C09139=1188.005,340.094,-74.713,-176.303,8.071,148.497
C09140=1188.000,340.372,-74.750,-176.301,8.074,148.497
C09141=1187.995,340.651,-74.787,-176.299,8.078,148.497
C09142=1187.991,340.929,-74.823,-176.296,8.081,148.498
C09143=1187.987,341.178,-74.856,-176.293,8.085,148.498
C09144=1187.982,341.425,-74.888,-176.291,8.088,148.498
C09145=1187.978,341.672,-74.921,-176.289,8.091,148.498
C09146=1187.974,341.921,-74.953,-176.287,8.094,148.498
C09147=1187.970,342.168,-74.987,-176.285,8.097,148.499
C09148=1187.966,342.416,-75.018,-176.283,8.101,148.499
C09149=1187.962,342.664,-75.052,-176.280,8.104,148.499
C09150=1187.958,342.912,-75.084,-176.278,8.107,148.499
C09151=1187.953,343.160,-75.117,-176.275,8.110,148.499
C09152=1187.950,343.408,-75.150,-176.273,8.114,148.499
C09153=1187.945,343.655,-75.182,-176.271,8.117,148.500
C09154=1187.941,343.903,-75.215,-176.269,8.120,148.500
C09155=1187.937,344.151,-75.248,-176.266,8.124,148.500
C09156=1187.932,344.399,-75.281,-176.264,8.127,148.500
C09157=1187.929,344.646,-75.313,-176.262,8.129,148.501
C09158=1187.925,344.894,-75.346,-176.260,8.133,148.501
C09159=1187.920,345.143,-75.379,-176.258,8.136,148.501
C09160=1187.916,345.390,-75.412,-176.256,8.139,148.501
C09161=1187.912,345.638,-75.445,-176.253,8.143,148.501
C09162=1187.909,345.885,-75.478,-176.251,8.146,148.502
C09163=1187.904,346.134,-75.510,-176.249,8.149,148.502
C09164=1187.900,346.382,-75.543,-176.247,8.153,148.502
C09165=1187.896,346.629,-75.576,-176.244,8.156,148.502
C09166=1187.892,346.877,-75.609,-176.242,8.159,148.502
C09167=1187.888,347.125,-75.643,-176.240,8.163,148.503
C09168=1187.883,347.373,-75.675,-176.238,8.165,148.503
C09169=1187.879,347.621,-75.708,-176.236,8.168,148.503
C09170=1187.876,347.868,-75.741,-176.234,8.172,148.503
C09171=1187.872,348.116,-75.774,-176.232,8.175,148.504
C09172=1187.867,348.364,-75.807,-176.229,8.178,148.504
C09173=1187.863,348.611,-75.840,-176.227,8.182,148.504
C09174=1187.859,348.859,-75.873,-176.225,8.185,148.504
C09175=1187.855,349.107,-75.907,-176.223,8.189,148.505
C09176=1187.851,349.355,-75.940,-176.221,8.192,148.505
C09177=1187.847,349.602,-75.973,-176.218,8.195,148.505
C09178=1187.842,349.851,-76.005,-176.216,8.199,148.505
C09179=1187.838,350.098,-76.038,-176.214,8.202,148.506
C09180=1187.834,350.346,-76.072,-176.212,8.205,148.506
C09181=1187.830,350.594,-76.105,-176.211,8.208,148.506
C09182=1187.826,350.842,-76.138,-176.208,8.211,148.506
C09183=1187.822,351.089,-76.171,-176.206,8.215,148.507
C09184=1187.818,351.336,-76.205,-176.204,8.218,148.507
C09185=1187.814,351.584,-76.238,-176.202,8.221,148.507
C09186=1187.809,351.832,-76.271,-176.200,8.225,148.507
C09187=1187.805,352.080,-76.304,-176.197,8.228,148.508
C09188=1187.801,352.327,-76.338,-176.195,8.232,148.508
C09189=1187.797,352.575,-76.371,-176.193,8.235,148.508
C09190=1187.793,352.824,-76.404,-176.191,8.238,148.508
C09191=1187.789,353.071,-76.437,-176.189,8.242,148.509
C09192=1187.785,353.319,-76.471,-176.187,8.245,148.509
C09193=1187.781,353.567,-76.504,-176.184,8.248,148.509
C09194=1187.777,353.814,-76.538,-176.183,8.251,148.510
C09195=1187.773,354.062,-76.571,-176.181,8.255,148.510
C09196=1187.768,354.310,-76.604,-176.179,8.258,148.510
C09197=1187.764,354.557,-76.638,-176.176,8.261,148.510
C09198=1187.760,354.805,-76.671,-176.175,8.265,148.511
C09199=1187.757,355.053,-76.705,-176.172,8.268,148.511
C09200=1187.753,355.301,-76.738,-176.170,8.272,148.511
C09201=1187.748,355.548,-76.771,-176.168,8.275,148.512
C09202=1187.744,355.796,-76.805,-176.166,8.278,148.512
C09203=1187.740,356.043,-76.838,-176.164,8.282,148.512
C09204=1187.736,356.291,-76.872,-176.162,8.285,148.512
C09205=1187.732,356.540,-76.906,-176.160,8.289,148.513
C09206=1187.728,356.787,-76.939,-176.158,8.292,148.513
C09207=1187.724,357.034,-76.973,-176.156,8.295,148.513
C09208=1187.720,357.282,-77.006,-176.154,8.298,148.513
C09209=1187.715,357.530,-77.040,-176.152,8.302,148.514
C09210=1187.711,357.777,-77.073,-176.150,8.305,148.514
C09211=1187.708,358.026,-77.107,-176.148,8.309,148.515
C09212=1187.704,358.273,-77.141,-176.146,8.312,148.515
C09213=1187.700,358.521,-77.174,-176.144,8.316,148.515
C09214=1187.695,358.769,-77.208,-176.142,8.319,148.515
C09215=1187.691,359.016,-77.242,-176.140,8.323,148.516
C09216=1187.687,359.264,-77.275,-176.138,8.326,148.516
C09217=1187.684,359.511,-77.309,-176.136,8.330,148.517
C09218=1187.679,359.759,-77.343,-176.134,8.333,148.517
C09219=1187.675,360.006,-77.377,-176.133,8.336,148.517
C09220=1187.671,360.255,-77.410,-176.131,8.339,148.518
C09221=1187.668,360.502,-77.444,-176.128,8.343,148.518
C09222=1187.663,360.750,-77.478,-176.127,8.346,148.518
C09223=1187.659,360.997,-77.512,-176.124,8.350,148.518
C09224=1187.655,361.246,-77.545,-176.123,8.353,148.519
C09225=1187.651,361.493,-77.580,-176.121,8.357,148.519
C09226=1187.647,361.741,-77.613,-176.119,8.359,148.520
C09227=1187.643,361.988,-77.647,-176.117,8.363,148.520
C09228=1187.639,362.236,-77.682,-176.116,8.367,148.520
C09229=1187.635,362.484,-77.715,-176.113,8.370,148.521
C09230=1187.631,362.731,-77.749,-176.111,8.374,148.521
C09231=1187.626,362.979,-77.782,-176.110,8.377,148.521
C09232=1187.623,363.227,-77.817,-176.108,8.380,148.522
C09233=1187.619,363.474,-77.850,-176.106,8.383,148.522
C09234=1187.614,363.722,-77.884,-176.104,8.387,148.523
C09235=1187.611,363.970,-77.918,-176.103,8.391,148.523
C09236=1187.606,364.217,-77.953,-176.101,8.394,148.523
C09237=1187.602,364.465,-77.986,-176.100,8.397,148.524
C09238=1187.599,364.713,-78.020,-176.098,8.401,148.524
C09239=1187.594,364.960,-78.055,-176.095,8.404,148.524
C09240=1187.590,365.208,-78.088,-176.094,8.408,148.525
C09241=1187.586,365.456,-78.123,-176.092,8.410,148.525
C09242=1187.582,365.703,-78.157,-176.091,8.414,148.526
C09243=1187.578,365.984,-78.195,-176.089,8.418,148.526
C09244=1187.573,366.265,-78.235,-176.086,8.422,148.527
C09245=1187.568,366.547,-78.273,-176.085,8.426,148.527
C09246=1187.564,366.828,-78.312,-176.083,8.429,148.527
C09247=1187.560,367.076,-78.345,-176.081,8.433,148.528
C09248=1187.556,367.323,-78.380,-176.079,8.437,148.528
C09249=1187.553,367.571,-78.414,-176.078,8.439,148.529
C09250=1187.548,367.819,-78.448,-176.076,8.443,148.529
C09251=1187.543,368.066,-78.482,-176.075,8.447,148.530
C09252=1187.540,368.314,-78.517,-176.074,8.450,148.530
C09253=1187.535,368.561,-78.551,-176.072,8.453,148.531
C09254=1187.532,368.809,-78.585,-176.070,8.457,148.531
C09255=1187.527,369.057,-78.620,-176.069,8.460,148.531
C09256=1187.524,369.304,-78.654,-176.067,8.463,148.532
C09257=1187.520,369.552,-78.688,-176.065,8.467,148.532
C09258=1187.516,369.799,-78.722,-176.064,8.470,148.533
C09259=1187.511,370.046,-78.757,-176.062,8.474,148.533
C09260=1187.508,370.295,-78.790,-176.061,8.477,148.534
C09261=1187.503,370.542,-78.825,-176.059,8.480,148.534
C09262=1187.499,370.790,-78.860,-176.058,8.484,148.535
C09263=1187.495,371.038,-78.893,-176.056,8.487,148.535
C09264=1187.491,371.286,-78.928,-176.055,8.490,148.536
C09265=1187.488,371.533,-78.962,-176.054,8.493,148.536
C09266=1187.483,371.780,-78.997,-176.052,8.497,148.536
C09267=1187.479,372.028,-79.031,-176.050,8.501,148.537
C09268=1187.475,372.275,-79.065,-176.049,8.504,148.537
C09269=1187.471,372.524,-79.100,-176.048,8.507,148.538
C09270=1187.467,372.770,-79.135,-176.046,8.510,148.538
C09271=1187.464,373.018,-79.170,-176.045,8.514,148.539
C09272=1187.459,373.266,-79.204,-176.044,8.517,148.539
C09273=1187.456,373.513,-79.238,-176.042,8.521,148.540
C09274=1187.451,373.761,-79.273,-176.041,8.523,148.540
C09275=1187.447,374.008,-79.307,-176.039,8.527,148.541
C09276=1187.443,374.256,-79.342,-176.039,8.530,148.541
C09277=1187.439,374.503,-79.376,-176.037,8.534,148.542
C09278=1187.435,374.752,-79.411,-176.036,8.537,148.542
C09279=1187.431,374.998,-79.446,-176.035,8.540,148.543
C09280=1187.428,375.246,-79.480,-176.033,8.544,148.543
C09281=1187.423,375.494,-79.515,-176.032,8.546,148.544
C09282=1187.419,375.742,-79.549,-176.031,8.550,148.544
C09283=1187.415,375.989,-79.583,-176.029,8.553,148.545
C09284=1187.411,376.237,-79.618,-176.029,8.556,148.545
C09285=1187.407,376.484,-79.653,-176.027,8.560,148.546
C09286=1187.403,376.732,-79.688,-176.026,8.563,148.546
C09287=1187.399,376.979,-79.722,-176.025,8.567,148.547
C09288=1187.395,377.227,-79.757,-176.023,8.570,148.547
C09289=1187.391,377.474,-79.792,-176.023,8.573,148.548
C09290=1187.387,377.722,-79.827,-176.021,8.576,148.548
C09291=1187.383,377.969,-79.861,-176.020,8.580,148.549
C09292=1187.379,378.217,-79.896,-176.019,8.583,148.550
C09293=1187.375,378.464,-79.931,-176.018,8.585,148.550
C09294=1187.371,378.712,-79.966,-176.017,8.589,148.551
C09295=1187.366,378.960,-80.000,-176.016,8.592,148.551
C09296=1187.363,379.207,-80.035,-176.015,8.595,148.552
C09297=1187.359,379.455,-80.070,-176.014,8.598,148.552
C09298=1187.355,379.702,-80.104,-176.012,8.602,148.553
C09299=1187.351,379.950,-80.139,-176.012,8.605,148.553
C09300=1187.347,380.197,-80.174,-176.011,8.608,148.554
C09301=1187.343,380.445,-80.209,-176.009,8.611,148.554
C09302=1187.339,380.692,-80.244,-176.009,8.614,148.555
C09303=1187.335,380.940,-80.279,-176.008,8.617,148.556
C09304=1187.331,381.187,-80.313,-176.007,8.621,148.556
C09305=1187.327,381.435,-80.349,-176.006,8.624,148.557
C09306=1187.322,381.682,-80.383,-176.004,8.627,148.557
C09307=1187.319,381.930,-80.419,-176.004,8.630,148.558
C09308=1187.315,382.178,-80.453,-176.003,8.633,148.558
C09309=1187.311,382.425,-80.487,-176.002,8.637,148.559
C09310=1187.307,382.673,-80.523,-176.001,8.640,148.559
C09311=1187.303,382.920,-80.557,-176.000,8.643,148.560
C09312=1187.299,383.167,-80.593,-176.000,8.646,148.561
C09313=1187.295,383.416,-80.628,-175.999,8.649,148.561
C09314=1187.291,383.662,-80.663,-175.998,8.652,148.562
C09315=1187.287,383.910,-80.698,-175.997,8.655,148.562
C09316=1187.283,384.157,-80.733,-175.996,8.658,148.563
C09317=1187.279,384.405,-80.767,-175.996,8.661,148.564
C09318=1187.276,384.653,-80.803,-175.995,8.664,148.564
C09319=1187.271,384.900,-80.837,-175.994,8.668,148.565
C09320=1187.267,385.148,-80.873,-175.993,8.671,148.565
C09321=1187.263,385.395,-80.907,-175.992,8.674,148.566
C09322=1187.259,385.642,-80.943,-175.992,8.677,148.566
C09323=1187.255,385.891,-80.978,-175.991,8.679,148.567
C09324=1187.251,386.137,-81.013,-175.991,8.682,148.568
C09325=1187.247,386.385,-81.048,-175.990,8.685,148.568
C09326=1187.243,386.632,-81.083,-175.989,8.688,148.569
C09327=1187.239,386.880,-81.118,-175.988,8.691,148.569
C09328=1187.235,387.128,-81.153,-175.988,8.694,148.570
C09329=1187.231,387.375,-81.188,-175.987,8.697,148.571
C09330=1187.227,387.623,-81.223,-175.987,8.700,148.571
C09331=1187.223,387.870,-81.259,-175.986,8.703,148.572
C09332=1187.219,388.118,-81.293,-175.986,8.706,148.572
C09333=1187.215,388.365,-81.329,-175.985,8.709,148.573
C09334=1187.211,388.613,-81.364,-175.984,8.712,148.574
C09335=1187.207,388.860,-81.399,-175.984,8.714,148.574
C09336=1187.203,389.108,-81.434,-175.983,8.717,148.575
C09337=1187.199,389.356,-81.469,-175.983,8.721,148.575
C09338=1187.195,389.603,-81.504,-175.982,8.723,148.576
C09339=1187.191,389.850,-81.540,-175.982,8.726,148.577
C09340=1187.187,390.098,-81.575,-175.981,8.729,148.577
C09341=1187.183,390.345,-81.610,-175.981,8.732,148.578
C09342=1187.179,390.592,-81.645,-175.980,8.735,148.578
C09343=1187.175,390.841,-81.680,-175.980,8.737,148.579
C09344=1187.171,391.087,-81.715,-175.979,8.740,148.580
C09345=1187.167,391.335,-81.751,-175.979,8.743,148.580
C09346=1187.164,391.582,-81.787,-175.978,8.746,148.581
C09347=1187.159,391.866,-81.827,-175.978,8.749,148.582
C09348=1187.155,392.150,-81.867,-175.978,8.751,148.582
C09349=1187.150,392.434,-81.907,-175.977,8.755,148.583
C09350=1187.145,392.717,-81.948,-175.977,8.758,148.584
C09351=1187.141,392.965,-81.983,-175.976,8.761,148.584
C09352=1187.137,393.212,-82.018,-175.976,8.764,148.585
C09353=1187.134,393.460,-82.054,-175.976,8.766,148.585
C09354=1187.129,393.706,-82.089,-175.975,8.769,148.586
C09355=1187.125,393.955,-82.124,-175.975,8.771,148.587
C09356=1187.122,394.202,-82.159,-175.974,8.775,148.587
C09357=1187.118,394.450,-82.195,-175.974,8.777,148.588
C09358=1187.114,394.696,-82.230,-175.974,8.779,148.588
C09359=1187.110,394.944,-82.265,-175.973,8.782,148.589
C09360=1187.106,395.192,-82.300,-175.973,8.785,148.590
C09361=1187.101,395.439,-82.336,-175.973,8.787,148.590
C09362=1187.097,395.687,-82.372,-175.973,8.790,148.591
C09363=1187.094,395.934,-82.407,-175.972,8.793,148.591
C09364=1187.090,396.182,-82.442,-175.973,8.795,148.592
C09365=1187.086,396.429,-82.477,-175.972,8.798,148.593
C09366=1187.082,396.676,-82.513,-175.972,8.800,148.593
C09367=1187.078,396.924,-82.548,-175.972,8.803,148.594
C09368=1187.074,397.171,-82.584,-175.971,8.805,148.595
C09369=1187.070,397.418,-82.619,-175.971,8.808,148.595
C09370=1187.066,397.667,-82.655,-175.971,8.810,148.596
C09371=1187.062,397.914,-82.690,-175.970,8.813,148.596
C09372=1187.058,398.161,-82.725,-175.970,8.816,148.597
C09373=1187.054,398.408,-82.761,-175.970,8.818,148.598
C09374=1187.050,398.656,-82.796,-175.970,8.820,148.598
C09375=1187.047,398.903,-82.832,-175.970,8.823,148.599
C09376=1187.042,399.150,-82.867,-175.970,8.825,148.599
C09377=1187.038,399.399,-82.903,-175.970,8.828,148.600
C09378=1187.034,399.646,-82.938,-175.969,8.831,148.600
C09379=1187.030,399.893,-82.973,-175.969,8.833,148.601
C09380=1187.026,400.141,-83.009,-175.969,8.835,148.602
C09381=1187.022,400.388,-83.044,-175.969,8.838,148.602
C09382=1187.019,400.636,-83.080,-175.968,8.840,148.603
C09383=1187.014,400.883,-83.116,-175.969,8.843,148.603
C09384=1187.010,401.130,-83.151,-175.968,8.845,148.604
C09385=1187.006,401.378,-83.187,-175.968,8.847,148.605
C09386=1187.003,401.625,-83.222,-175.968,8.850,148.605
C09387=1186.999,401.873,-83.257,-175.968,8.852,148.606
C09388=1186.994,402.120,-83.293,-175.968,8.854,148.606
C09389=1186.990,402.368,-83.329,-175.968,8.857,148.607
C09390=1186.986,402.615,-83.364,-175.968,8.859,148.608
C09391=1186.983,402.863,-83.400,-175.968,8.861,148.608
C09392=1186.979,403.110,-83.435,-175.967,8.864,148.609
C09393=1186.975,403.357,-83.470,-175.967,8.866,148.609
C09394=1186.970,403.605,-83.506,-175.967,8.868,148.610
C09395=1186.967,403.852,-83.542,-175.967,8.871,148.610
C09396=1186.963,404.099,-83.577,-175.967,8.873,148.611
C09397=1186.959,404.347,-83.613,-175.967,8.876,148.612
C09398=1186.954,404.595,-83.649,-175.967,8.878,148.612
C09399=1186.951,404.842,-83.684,-175.966,8.880,148.613
C09400=1186.947,405.090,-83.720,-175.967,8.883,148.613
C09401=1186.943,405.336,-83.755,-175.967,8.884,148.614
C09402=1186.939,405.584,-83.791,-175.967,8.886,148.614
C09403=1186.935,405.832,-83.827,-175.966,8.889,148.615
C09404=1186.931,406.079,-83.862,-175.967,8.891,148.616
C09405=1186.927,406.326,-83.898,-175.966,8.893,148.616
C09406=1186.923,406.573,-83.933,-175.966,8.896,148.617
C09407=1186.919,406.821,-83.969,-175.966,8.898,148.617
C09408=1186.915,407.069,-84.005,-175.967,8.900,148.618
C09409=1186.912,407.316,-84.040,-175.966,8.902,148.618
C09410=1186.907,407.563,-84.076,-175.966,8.904,148.619
C09411=1186.903,407.811,-84.112,-175.966,8.906,148.619
C09412=1186.899,408.058,-84.147,-175.966,8.909,148.620
C09413=1186.896,408.306,-84.183,-175.966,8.911,148.621
C09414=1186.892,408.553,-84.218,-175.966,8.913,148.621
C09415=1186.887,408.801,-84.254,-175.966,8.915,148.622
C09416=1186.883,409.048,-84.290,-175.965,8.917,148.622
C09417=1186.880,409.296,-84.325,-175.966,8.920,148.623
C09418=1186.876,409.542,-84.361,-175.966,8.921,148.623
C09419=1186.872,409.790,-84.398,-175.966,8.924,148.624
C09420=1186.868,410.038,-84.433,-175.965,8.926,148.624
C09421=1186.864,410.285,-84.468,-175.965,8.928,148.625
C09422=1186.860,410.532,-84.504,-175.966,8.930,148.625
C09423=1186.856,410.780,-84.540,-175.966,8.932,148.626
C09424=1186.852,411.027,-84.576,-175.965,8.934,148.627
C09425=1186.848,411.275,-84.611,-175.965,8.937,148.627
C09426=1186.843,411.522,-84.647,-175.965,8.938,148.628
C09427=1186.840,411.769,-84.682,-175.965,8.940,148.628
C09428=1186.836,412.017,-84.718,-175.965,8.943,148.629
C09429=1186.832,412.264,-84.754,-175.966,8.944,148.629
C09430=1186.828,412.512,-84.790,-175.965,8.947,148.630
C09431=1186.825,412.759,-84.826,-175.965,8.949,148.630
C09432=1186.820,413.006,-84.861,-175.966,8.950,148.631
C09433=1186.816,413.254,-84.897,-175.965,8.953,148.631
C09434=1186.812,413.501,-84.933,-175.965,8.955,148.632
C09435=1186.809,413.749,-84.968,-175.965,8.957,148.632
C09436=1186.804,413.997,-85.005,-175.965,8.958,148.633
C09437=1186.801,414.244,-85.040,-175.965,8.961,148.633
C09438=1186.797,414.490,-85.076,-175.965,8.962,148.634
C09439=1186.793,414.738,-85.112,-175.965,8.964,148.634
C09440=1186.789,414.986,-85.148,-175.965,8.967,148.635
C09441=1186.785,415.233,-85.183,-175.965,8.968,148.636
C09442=1186.781,415.481,-85.219,-175.965,8.971,148.636
C09443=1186.774,415.892,-85.279,-175.965,8.974,148.637
C09444=1186.770,416.304,-85.338,-175.965,8.977,148.638
C09445=1186.770,416.715,-85.397,-175.964,8.980,148.638
C09446=1186.774,417.125,-85.456,-175.965,8.983,148.639
C09447=1186.353,417.127,-85.497,-175.968,8.994,148.643
C09448=1186.349,416.714,-85.438,-175.968,8.991,148.642
C09449=1186.349,416.299,-85.379,-175.968,8.988,148.641
C09450=1186.353,415.883,-85.319,-175.968,8.985,148.640
C09451=1186.360,415.469,-85.259,-175.968,8.981,148.640
C09452=1186.363,415.222,-85.223,-175.968,8.979,148.639
C09453=1186.368,414.974,-85.187,-175.968,8.978,148.639
C09454=1186.371,414.727,-85.151,-175.968,8.975,148.638
C09455=1186.375,414.480,-85.116,-175.968,8.974,148.638
C09456=1186.380,414.232,-85.080,-175.968,8.971,148.637
C09457=1186.383,413.985,-85.044,-175.968,8.969,148.636
C09458=1186.387,413.737,-85.008,-175.968,8.968,148.636
C09459=1186.391,413.490,-84.972,-175.968,8.965,148.636
C09460=1186.395,413.243,-84.936,-175.968,8.963,148.635
C09461=1186.399,412.996,-84.901,-175.968,8.962,148.635
C09462=1186.403,412.748,-84.865,-175.968,8.959,148.634
C09463=1186.407,412.501,-84.829,-175.968,8.957,148.633
C09464=1186.411,412.253,-84.794,-175.968,8.956,148.633
C09465=1186.414,412.006,-84.758,-175.968,8.953,148.632
C09466=1186.419,411.758,-84.722,-175.968,8.951,148.632
C09467=1186.423,411.511,-84.687,-175.969,8.949,148.631
C09468=1186.427,411.264,-84.651,-175.968,8.947,148.631
C09469=1186.431,411.016,-84.614,-175.968,8.945,148.630
C09470=1186.435,410.769,-84.579,-175.969,8.943,148.630
C09471=1186.438,410.521,-84.543,-175.968,8.941,148.629
C09472=1186.443,410.274,-84.507,-175.968,8.939,148.629
C09473=1186.447,410.027,-84.472,-175.969,8.936,148.628
C09474=1186.451,409.779,-84.436,-175.969,8.934,148.628
C09475=1186.454,409.532,-84.401,-175.968,8.933,148.627
C09476=1186.459,409.284,-84.365,-175.969,8.931,148.627
C09477=1186.462,409.036,-84.329,-175.969,8.928,148.626
C09478=1186.466,408.790,-84.294,-175.969,8.926,148.625
C09479=1186.470,408.542,-84.258,-175.968,8.924,148.625
C09480=1186.475,408.294,-84.222,-175.969,8.922,148.624
C09481=1186.478,408.047,-84.186,-175.969,8.920,148.624
C09482=1186.482,407.800,-84.150,-175.969,8.917,148.623
C09483=1186.486,407.553,-84.115,-175.969,8.915,148.623
C09484=1186.490,407.305,-84.079,-175.969,8.913,148.622
C09485=1186.494,407.058,-84.044,-175.969,8.911,148.622
C09486=1186.498,406.810,-84.008,-175.969,8.909,148.621
C09487=1186.501,406.563,-83.972,-175.969,8.906,148.620
C09488=1186.506,406.316,-83.937,-175.969,8.904,148.620
C09489=1186.510,406.068,-83.901,-175.970,8.902,148.619
C09490=1186.514,405.821,-83.866,-175.969,8.900,148.619
C09491=1186.517,405.573,-83.830,-175.969,8.898,148.618
C09492=1186.522,405.325,-83.794,-175.969,8.896,148.618
C09493=1186.526,405.079,-83.759,-175.970,8.893,148.617
C09494=1186.530,404.831,-83.723,-175.969,8.891,148.616
C09495=1186.533,404.584,-83.688,-175.970,8.888,148.616
C09496=1186.537,404.336,-83.652,-175.970,8.886,148.615
C09497=1186.541,404.088,-83.616,-175.970,8.884,148.615
C09498=1186.546,403.842,-83.581,-175.970,8.881,148.614
C09499=1186.549,403.594,-83.545,-175.970,8.879,148.614
C09500=1186.553,403.346,-83.510,-175.970,8.877,148.613
C09501=1186.557,403.099,-83.474,-175.970,8.874,148.612
C09502=1186.562,402.852,-83.438,-175.970,8.873,148.612
C09503=1186.565,402.604,-83.403,-175.970,8.871,148.611
C09504=1186.569,402.357,-83.367,-175.970,8.868,148.611
C09505=1186.573,402.109,-83.332,-175.970,8.866,148.610
C09506=1186.578,401.862,-83.296,-175.971,8.863,148.609
C09507=1186.581,401.614,-83.261,-175.970,8.861,148.609
C09508=1186.585,401.367,-83.226,-175.971,8.859,148.608
C09509=1186.589,401.119,-83.190,-175.972,8.856,148.608
C09510=1186.592,400.872,-83.154,-175.971,8.853,148.607
C09511=1186.597,400.625,-83.119,-175.972,8.851,148.606
C09512=1186.601,400.377,-83.083,-175.972,8.848,148.606
C09513=1186.605,400.130,-83.048,-175.972,8.846,148.605
C09514=1186.608,399.882,-83.012,-175.972,8.844,148.605
C09515=1186.613,399.635,-82.977,-175.972,8.841,148.604
C09516=1186.616,399.388,-82.941,-175.972,8.839,148.603
C09517=1186.620,399.140,-82.906,-175.972,8.837,148.603
C09518=1186.625,398.892,-82.870,-175.972,8.834,148.602
C09519=1186.629,398.645,-82.835,-175.972,8.832,148.602
C09520=1186.633,398.398,-82.800,-175.973,8.829,148.601
C09521=1186.636,398.150,-82.764,-175.973,8.826,148.601
C09522=1186.640,397.903,-82.729,-175.973,8.824,148.600
C09523=1186.644,397.656,-82.693,-175.973,8.821,148.599
C09524=1186.649,397.408,-82.657,-175.974,8.819,148.599
C09525=1186.652,397.160,-82.622,-175.973,8.817,148.598
C09526=1186.657,396.913,-82.587,-175.974,8.814,148.597
C09527=1186.661,396.665,-82.552,-175.975,8.811,148.597
C09528=1186.664,396.418,-82.516,-175.974,8.809,148.596
C09529=1186.668,396.170,-82.481,-175.975,8.806,148.596
C09530=1186.672,395.924,-82.445,-175.975,8.803,148.595
C09531=1186.676,395.676,-82.411,-175.975,8.801,148.594
C09532=1186.681,395.428,-82.374,-175.975,8.799,148.594
C09533=1186.685,395.181,-82.339,-175.976,8.795,148.593
C09534=1186.688,394.933,-82.304,-175.976,8.793,148.593
C09535=1186.692,394.686,-82.268,-175.976,8.791,148.592
C09536=1186.696,394.438,-82.233,-175.977,8.787,148.591
C09537=1186.700,394.191,-82.198,-175.977,8.785,148.591
C09538=1186.704,393.944,-82.163,-175.977,8.783,148.590
C09539=1186.708,393.696,-82.127,-175.978,8.780,148.590
C09540=1186.712,393.449,-82.092,-175.978,8.777,148.589
C09541=1186.716,393.201,-82.057,-175.978,8.775,148.588
C09542=1186.720,392.954,-82.021,-175.979,8.772,148.588
C09543=1186.723,392.706,-81.986,-175.979,8.769,148.587
C09544=1186.728,392.422,-81.946,-175.980,8.766,148.586
C09545=1186.732,392.139,-81.905,-175.980,8.763,148.586
C09546=1186.737,391.855,-81.865,-175.981,8.759,148.585
C09547=1186.742,391.571,-81.824,-175.981,8.756,148.584
C09548=1186.746,391.325,-81.789,-175.981,8.754,148.584
C09549=1186.750,391.076,-81.754,-175.982,8.751,148.583
C09550=1186.754,390.829,-81.718,-175.982,8.748,148.582
C09551=1186.758,390.582,-81.683,-175.983,8.745,148.582
C09552=1186.762,390.334,-81.648,-175.983,8.743,148.581
C09553=1186.766,390.086,-81.612,-175.984,8.740,148.581
C09554=1186.770,389.839,-81.577,-175.984,8.737,148.580
C09555=1186.774,389.591,-81.542,-175.984,8.734,148.579
C09556=1186.778,389.344,-81.507,-175.985,8.731,148.579
C09557=1186.782,389.097,-81.472,-175.985,8.729,148.578
C09558=1186.786,388.849,-81.437,-175.986,8.725,148.578
C09559=1186.790,388.601,-81.401,-175.987,8.722,148.577
C09560=1186.794,388.355,-81.366,-175.987,8.720,148.576
C09561=1186.798,388.106,-81.331,-175.988,8.717,148.576
C09562=1186.802,387.859,-81.296,-175.989,8.714,148.575
C09563=1186.806,387.612,-81.261,-175.988,8.711,148.575
C09564=1186.810,387.364,-81.226,-175.989,8.708,148.574
C09565=1186.814,387.117,-81.190,-175.990,8.705,148.573
C09566=1186.818,386.869,-81.156,-175.991,8.702,148.573
C09567=1186.821,386.622,-81.121,-175.991,8.700,148.572
C09568=1186.825,386.374,-81.086,-175.992,8.696,148.572
C09569=1186.829,386.127,-81.051,-175.993,8.693,148.571
C09570=1186.833,385.879,-81.015,-175.993,8.690,148.571
C09571=1186.838,385.632,-80.981,-175.994,8.687,148.570
C09572=1186.841,385.385,-80.945,-175.995,8.684,148.569
C09573=1186.845,385.136,-80.910,-175.995,8.681,148.569
C09574=1186.849,384.890,-80.875,-175.996,8.678,148.568
C09575=1186.853,384.642,-80.840,-175.996,8.675,148.567
C09576=1186.857,384.394,-80.805,-175.997,8.672,148.567
C09577=1186.862,384.147,-80.770,-175.998,8.669,148.566
C09578=1186.865,383.899,-80.735,-175.999,8.666,148.566
C09579=1186.870,383.652,-80.700,-176.000,8.663,148.565
C09580=1186.874,383.404,-80.665,-176.001,8.660,148.565
C09581=1186.878,383.156,-80.630,-176.001,8.657,148.564
C09582=1186.881,382.910,-80.595,-176.002,8.654,148.563
C09583=1186.885,382.661,-80.561,-176.003,8.651,148.563
C09584=1186.889,382.415,-80.525,-176.004,8.648,148.562
C09585=1186.893,382.167,-80.491,-176.005,8.645,148.562
C09586=1186.898,381.919,-80.456,-176.006,8.642,148.561
C09587=1186.902,381.672,-80.421,-176.007,8.638,148.561
C09588=1186.905,381.423,-80.386,-176.008,8.635,148.560
C09589=1186.910,381.177,-80.351,-176.009,8.631,148.559
C09590=1186.913,380.929,-80.316,-176.010,8.628,148.559
C09591=1186.918,380.681,-80.282,-176.011,8.626,148.558
C09592=1186.921,380.434,-80.246,-176.012,8.622,148.558
C09593=1186.926,380.187,-80.212,-176.012,8.619,148.557
C09594=1186.929,379.939,-80.176,-176.014,8.615,148.557
C09595=1186.933,379.691,-80.141,-176.015,8.612,148.556
C09596=1186.937,379.444,-80.108,-176.016,8.610,148.556
C09597=1186.941,379.196,-80.072,-176.017,8.606,148.555
C09598=1186.945,378.949,-80.038,-176.018,8.603,148.554
C09599=1186.949,378.701,-80.003,-176.019,8.599,148.554
C09600=1186.954,378.454,-79.968,-176.020,8.597,148.554
C09601=1186.957,378.206,-79.933,-176.021,8.594,148.553
C09602=1186.962,377.959,-79.899,-176.022,8.590,148.552
C09603=1186.965,377.711,-79.864,-176.024,8.587,148.552
C09604=1186.970,377.464,-79.829,-176.024,8.584,148.551
C09605=1186.974,377.216,-79.794,-176.026,8.580,148.551
C09606=1186.978,376.969,-79.760,-176.027,8.577,148.550
C09607=1186.982,376.720,-79.725,-176.028,8.574,148.550
C09608=1186.986,376.474,-79.690,-176.030,8.570,148.549
C09609=1186.990,376.226,-79.655,-176.030,8.567,148.549
C09610=1186.994,375.978,-79.621,-176.032,8.564,148.548
C09611=1186.998,375.730,-79.587,-176.033,8.560,148.548
C09612=1187.002,375.483,-79.552,-176.034,8.557,148.547
C09613=1187.005,375.236,-79.517,-176.036,8.554,148.547
C09614=1187.010,374.988,-79.483,-176.036,8.551,148.546
C09615=1187.014,374.740,-79.448,-176.038,8.547,148.546
C09616=1187.018,374.493,-79.413,-176.039,8.544,148.545
C09617=1187.021,374.245,-79.379,-176.040,8.541,148.545
C09618=1187.026,373.998,-79.345,-176.042,8.538,148.544
C09619=1187.030,373.750,-79.309,-176.043,8.534,148.544
C09620=1187.033,373.503,-79.275,-176.045,8.531,148.543
C09621=1187.037,373.255,-79.240,-176.045,8.528,148.543
C09622=1187.042,373.007,-79.206,-176.047,8.524,148.542
C09623=1187.045,372.760,-79.172,-176.049,8.521,148.542
C09624=1187.050,372.512,-79.137,-176.050,8.517,148.541
C09625=1187.054,372.265,-79.103,-176.052,8.514,148.541
C09626=1187.058,372.017,-79.069,-176.053,8.511,148.540
C09627=1187.062,371.770,-79.034,-176.054,8.507,148.540
C09628=1187.065,371.522,-79.000,-176.056,8.504,148.539
C09629=1187.070,371.274,-78.965,-176.057,8.501,148.539
C09630=1187.074,371.026,-78.931,-176.058,8.497,148.538
C09631=1187.078,370.779,-78.897,-176.060,8.494,148.538
C09632=1187.082,370.532,-78.862,-176.062,8.490,148.537
C09633=1187.086,370.284,-78.828,-176.063,8.487,148.537
C09634=1187.090,370.036,-78.793,-176.065,8.484,148.537
C09635=1187.094,369.788,-78.759,-176.066,8.481,148.536
C09636=1187.098,369.541,-78.725,-176.067,8.477,148.536
C09637=1187.102,369.294,-78.690,-176.069,8.473,148.535
C09638=1187.106,369.046,-78.656,-176.070,8.471,148.535
C09639=1187.110,368.799,-78.622,-176.072,8.467,148.534
C09640=1187.114,368.551,-78.587,-176.074,8.463,148.534
C09641=1187.118,368.303,-78.553,-176.075,8.461,148.534
C09642=1187.122,368.056,-78.520,-176.077,8.457,148.533
C09643=1187.126,367.807,-78.485,-176.079,8.453,148.533
C09644=1187.130,367.560,-78.451,-176.080,8.449,148.532
C09645=1187.135,367.313,-78.417,-176.082,8.447,148.532
C09646=1187.138,367.065,-78.382,-176.083,8.443,148.531
C09647=1187.142,366.818,-78.348,-176.085,8.439,148.531
C09648=1187.147,366.536,-78.310,-176.087,8.436,148.530
C09649=1187.151,366.254,-78.271,-176.089,8.432,148.530
C09650=1187.156,365.973,-78.232,-176.091,8.429,148.529
C09651=1187.161,365.692,-78.193,-176.093,8.424,148.529
C09652=1187.164,365.445,-78.159,-176.094,8.421,148.529
C09653=1187.169,365.196,-78.125,-176.096,8.418,148.528
C09654=1187.173,364.949,-78.091,-176.098,8.414,148.528
C09655=1187.177,364.702,-78.057,-176.100,8.411,148.528
C09656=1187.180,364.454,-78.022,-176.102,8.407,148.527
C09657=1187.185,364.206,-77.989,-176.103,8.404,148.527
C09658=1187.189,363.959,-77.955,-176.105,8.401,148.526
C09659=1187.192,363.711,-77.921,-176.107,8.397,148.526
C09660=1187.197,363.463,-77.887,-176.109,8.393,148.525
C09661=1187.201,363.216,-77.853,-176.111,8.390,148.525
C09662=1187.205,362.969,-77.819,-176.112,8.387,148.525
C09663=1187.209,362.720,-77.785,-176.114,8.384,148.524
C09664=1187.213,362.473,-77.751,-176.116,8.380,148.524
C09665=1187.217,362.225,-77.718,-176.118,8.377,148.524
C09666=1187.221,361.977,-77.683,-176.120,8.373,148.523
C09667=1187.225,361.730,-77.649,-176.121,8.369,148.523
C09668=1187.229,361.482,-77.616,-176.123,8.367,148.523
C09669=1187.234,361.235,-77.582,-176.125,8.363,148.522
C09670=1187.237,360.986,-77.548,-176.127,8.360,148.522
C09671=1187.241,360.739,-77.514,-176.129,8.356,148.522
C09672=1187.246,360.491,-77.480,-176.131,8.353,148.521
C09673=1187.250,360.244,-77.447,-176.133,8.349,148.521
C09674=1187.253,359.996,-77.413,-176.135,8.346,148.520
C09675=1187.258,359.748,-77.379,-176.137,8.342,148.520
C09676=1187.262,359.501,-77.345,-176.138,8.340,148.520
C09677=1187.266,359.253,-77.312,-176.140,8.336,148.519
C09678=1187.269,359.005,-77.278,-176.142,8.333,148.519
C09679=1187.274,358.758,-77.244,-176.144,8.329,148.519
C09680=1187.278,358.510,-77.210,-176.146,8.326,148.519
C09681=1187.282,358.262,-77.177,-176.148,8.322,148.518
C09682=1187.286,358.015,-77.143,-176.151,8.319,148.518
C09683=1187.290,357.766,-77.109,-176.152,8.315,148.517
C09684=1187.294,357.519,-77.075,-176.155,8.312,148.517
C09685=1187.298,357.271,-77.042,-176.156,8.308,148.517
C09686=1187.302,357.024,-77.009,-176.159,8.305,148.517
C09687=1187.306,356.777,-76.975,-176.161,8.302,148.516
C09688=1187.310,356.528,-76.942,-176.163,8.298,148.516
C09689=1187.315,356.280,-76.908,-176.165,8.295,148.516
C09690=1187.318,356.033,-76.874,-176.167,8.292,148.516
C09691=1187.323,355.785,-76.841,-176.168,8.289,148.515
C09692=1187.327,355.538,-76.808,-176.171,8.285,148.515
C09693=1187.331,355.290,-76.775,-176.172,8.282,148.514
C09694=1187.335,355.043,-76.741,-176.175,8.278,148.514
C09695=1187.339,354.794,-76.707,-176.177,8.275,148.514
C09696=1187.343,354.546,-76.673,-176.179,8.271,148.514
C09697=1187.347,354.299,-76.640,-176.181,8.268,148.513
C09698=1187.351,354.051,-76.606,-176.183,8.265,148.513
C09699=1187.355,353.804,-76.573,-176.186,8.261,148.513
C09700=1187.359,353.556,-76.540,-176.187,8.258,148.512
C09701=1187.363,353.308,-76.507,-176.190,8.254,148.512
C09702=1187.368,353.060,-76.474,-176.192,8.251,148.512
C09703=1187.371,352.812,-76.440,-176.194,8.248,148.512
C09704=1187.375,352.564,-76.407,-176.196,8.244,148.511
C09705=1187.379,352.317,-76.373,-176.198,8.241,148.511
C09706=1187.383,352.069,-76.340,-176.200,8.238,148.511
C09707=1187.387,351.822,-76.307,-176.202,8.235,148.511
C09708=1187.392,351.574,-76.273,-176.204,8.231,148.510
C09709=1187.396,351.326,-76.240,-176.206,8.228,148.510
C09710=1187.401,351.078,-76.207,-176.208,8.225,148.510
C09711=1187.405,350.831,-76.174,-176.211,8.221,148.510
C09712=1187.409,350.583,-76.141,-176.213,8.218,148.509
C09713=1187.413,350.335,-76.107,-176.215,8.215,148.509
C09714=1187.417,350.087,-76.074,-176.217,8.211,148.509
C09715=1187.420,349.840,-76.042,-176.219,8.208,148.509
C09716=1187.425,349.592,-76.009,-176.221,8.205,148.508
C09717=1187.429,349.344,-75.975,-176.224,8.201,148.508
C09718=1187.433,349.097,-75.942,-176.226,8.198,148.508
C09719=1187.437,348.849,-75.909,-176.228,8.195,148.508
C09720=1187.441,348.601,-75.876,-176.230,8.192,148.507
C09721=1187.445,348.353,-75.842,-176.232,8.189,148.507
C09722=1187.449,348.104,-75.810,-176.234,8.185,148.507
C09723=1187.453,347.857,-75.777,-176.236,8.182,148.507
C09724=1187.457,347.609,-75.744,-176.238,8.178,148.506
C09725=1187.462,347.361,-75.710,-176.241,8.175,148.506
C09726=1187.466,347.114,-75.678,-176.243,8.172,148.506
C09727=1187.470,346.867,-75.645,-176.245,8.169,148.506
C09728=1187.474,346.619,-75.612,-176.247,8.165,148.506
C09729=1187.478,346.371,-75.580,-176.250,8.162,148.505
C09730=1187.482,346.123,-75.546,-176.252,8.159,148.505
C09731=1187.487,345.875,-75.513,-176.254,8.155,148.505
C09732=1187.491,345.628,-75.480,-176.256,8.152,148.505
C09733=1187.495,345.379,-75.448,-176.258,8.149,148.504
C09734=1187.499,345.132,-75.414,-176.260,8.146,148.504
C09735=1187.503,344.884,-75.382,-176.263,8.143,148.504
C09736=1187.507,344.636,-75.349,-176.265,8.139,148.504
C09737=1187.511,344.388,-75.316,-176.267,8.136,148.504
C09738=1187.515,344.140,-75.283,-176.269,8.133,148.503
C09739=1187.520,343.893,-75.250,-176.272,8.130,148.503
C09740=1187.523,343.645,-75.218,-176.274,8.126,148.503
C09741=1187.527,343.397,-75.185,-176.276,8.123,148.503
C09742=1187.532,343.149,-75.152,-176.278,8.120,148.502
C09743=1187.536,342.901,-75.119,-176.281,8.117,148.502
C09744=1187.540,342.654,-75.087,-176.283,8.113,148.502
C09745=1187.544,342.406,-75.054,-176.285,8.111,148.502
C09746=1187.549,342.158,-75.022,-176.287,8.107,148.502
C09747=1187.553,341.910,-74.988,-176.290,8.104,148.502
C09748=1187.556,341.662,-74.957,-176.292,8.101,148.501
C09749=1187.561,341.414,-74.923,-176.294,8.097,148.501
C09750=1187.565,341.166,-74.891,-176.296,8.094,148.501
C09751=1187.569,340.918,-74.858,-176.299,8.091,148.501
C09752=1187.574,340.640,-74.821,-176.301,8.088,148.501
C09753=1187.578,340.361,-74.785,-176.304,8.084,148.501
C09754=1187.583,340.082,-74.749,-176.306,8.080,148.500
C09755=1187.587,339.803,-74.712,-176.309,8.076,148.500
C09756=1187.591,339.556,-74.679,-176.311,8.074,148.500
C09757=1187.596,339.308,-74.647,-176.313,8.071,148.500
C09758=1187.600,339.060,-74.615,-176.316,8.067,148.500
C09759=1187.604,338.812,-74.582,-176.318,8.064,148.499
C09760=1187.609,338.564,-74.550,-176.320,8.061,148.499
C09761=1187.612,338.317,-74.517,-176.322,8.057,148.499
C09762=1187.617,338.068,-74.485,-176.325,8.054,148.499
C09763=1187.621,337.821,-74.453,-176.327,8.051,148.499
C09764=1187.625,337.573,-74.420,-176.330,8.048,148.499
C09765=1187.629,337.325,-74.388,-176.332,8.044,148.498
C09766=1187.633,337.077,-74.356,-176.334,8.041,148.498
C09767=1187.637,336.829,-74.323,-176.336,8.039,148.498
C09768=1187.642,336.582,-74.291,-176.339,8.036,148.498
C09769=1187.646,336.333,-74.259,-176.341,8.032,148.498
C09770=1187.649,336.086,-74.226,-176.344,8.029,148.498
C09771=1187.654,335.838,-74.194,-176.346,8.026,148.498
C09772=1187.658,335.590,-74.162,-176.348,8.023,148.497
C09773=1187.663,335.342,-74.130,-176.350,8.019,148.497
C09774=1187.666,335.094,-74.097,-176.353,8.016,148.497
C09775=1187.670,334.846,-74.065,-176.355,8.013,148.497
C09776=1187.674,334.598,-74.033,-176.357,8.010,148.497
C09777=1187.679,334.350,-74.001,-176.360,8.007,148.497
C09778=1187.683,334.102,-73.969,-176.362,8.004,148.497
C09779=1187.687,333.855,-73.936,-176.364,8.001,148.496
C09780=1187.691,333.607,-73.904,-176.367,7.998,148.496
C09781=1187.695,333.359,-73.872,-176.369,7.994,148.496
C09782=1187.700,333.111,-73.840,-176.371,7.991,148.496
C09783=1187.703,332.863,-73.808,-176.374,7.988,148.496
C09784=1187.708,332.615,-73.776,-176.376,7.985,148.496
C09785=1187.712,332.367,-73.744,-176.379,7.981,148.495
C09786=1187.716,332.119,-73.712,-176.381,7.979,148.495
C09787=1187.720,331.871,-73.680,-176.383,7.976,148.495
C09788=1187.724,331.624,-73.648,-176.385,7.973,148.495
C09789=1187.729,331.375,-73.616,-176.388,7.970,148.495
C09790=1187.732,331.128,-73.583,-176.390,7.966,148.495
C09791=1187.737,330.880,-73.552,-176.392,7.963,148.495
C09792=1187.741,330.632,-73.520,-176.395,7.960,148.495
C09793=1187.745,330.383,-73.488,-176.397,7.957,148.494
C09794=1187.749,330.136,-73.457,-176.400,7.954,148.494
C09795=1187.754,329.888,-73.424,-176.402,7.951,148.494
C09796=1187.758,329.640,-73.393,-176.404,7.948,148.494
C09797=1187.762,329.392,-73.361,-176.407,7.945,148.494
C09798=1187.766,329.144,-73.329,-176.409,7.942,148.494
C09799=1187.771,328.897,-73.297,-176.412,7.939,148.494
C09800=1187.774,328.649,-73.265,-176.414,7.935,148.494
C09801=1187.779,328.400,-73.233,-176.417,7.932,148.494
C09802=1187.783,328.153,-73.201,-176.419,7.929,148.493
C09803=1187.787,327.905,-73.170,-176.422,7.926,148.493
C09804=1187.791,327.656,-73.139,-176.423,7.923,148.493
C09805=1187.796,327.409,-73.106,-176.425,7.920,148.493
C09806=1187.800,327.161,-73.075,-176.428,7.917,148.493
C09807=1187.804,326.913,-73.043,-176.430,7.914,148.493
C09808=1187.808,326.665,-73.011,-176.433,7.911,148.493
C09809=1187.812,326.416,-72.980,-176.435,7.907,148.493
C09810=1187.817,326.169,-72.948,-176.438,7.904,148.493
C09811=1187.820,325.921,-72.916,-176.440,7.901,148.492
C09812=1187.825,325.673,-72.885,-176.442,7.899,148.492
C09813=1187.829,325.425,-72.854,-176.445,7.896,148.492
C09814=1187.833,325.177,-72.822,-176.447,7.893,148.492
C09815=1187.837,324.929,-72.790,-176.450,7.889,148.492
C09816=1187.841,324.681,-72.758,-176.452,7.886,148.492
C09817=1187.846,324.433,-72.727,-176.455,7.883,148.492
C09818=1187.849,324.185,-72.695,-176.457,7.880,148.492
C09819=1187.854,323.938,-72.664,-176.460,7.877,148.492
C09820=1187.858,323.689,-72.633,-176.462,7.874,148.492
C09821=1187.862,323.442,-72.601,-176.464,7.871,148.492
C09822=1187.866,323.193,-72.570,-176.467,7.868,148.492
C09823=1187.870,322.946,-72.539,-176.469,7.865,148.492
C09824=1187.874,322.698,-72.507,-176.472,7.862,148.491
C09825=1187.879,322.449,-72.475,-176.474,7.859,148.491
C09826=1187.883,322.201,-72.443,-176.477,7.855,148.491
C09827=1187.888,321.953,-72.413,-176.479,7.853,148.491
C09828=1187.891,321.705,-72.381,-176.481,7.850,148.491
C09829=1187.896,321.457,-72.350,-176.484,7.847,148.491
C09830=1187.900,321.209,-72.318,-176.486,7.844,148.491
C09831=1187.904,320.961,-72.288,-176.489,7.841,148.491
C09832=1187.908,320.713,-72.256,-176.491,7.838,148.491
C09833=1187.913,320.465,-72.225,-176.494,7.834,148.491
C09834=1187.916,320.217,-72.193,-176.496,7.832,148.491
C09835=1187.921,319.969,-72.162,-176.498,7.829,148.491
C09836=1187.925,319.721,-72.130,-176.501,7.826,148.490
C09837=1187.929,319.473,-72.100,-176.503,7.823,148.490
C09838=1187.933,319.225,-72.069,-176.506,7.819,148.490
C09839=1187.938,318.977,-72.037,-176.508,7.816,148.490
C09840=1187.942,318.729,-72.006,-176.511,7.813,148.490
C09841=1187.946,318.481,-71.974,-176.513,7.811,148.490
C09842=1187.951,318.234,-71.944,-176.515,7.808,148.490
C09843=1187.954,317.985,-71.913,-176.518,7.805,148.490
C09844=1187.958,317.738,-71.882,-176.520,7.802,148.490
C09845=1187.962,317.489,-71.851,-176.523,7.799,148.490
C09846=1187.967,317.241,-71.820,-176.525,7.795,148.490
C09847=1187.971,316.993,-71.789,-176.528,7.792,148.490
C09848=1187.975,316.745,-71.757,-176.530,7.790,148.490
C09849=1187.980,316.497,-71.726,-176.532,7.787,148.490
C09850=1187.984,316.249,-71.695,-176.535,7.784,148.490
C09851=1187.988,316.001,-71.664,-176.538,7.781,148.490
C09852=1187.992,315.754,-71.634,-176.540,7.777,148.489
C09853=1187.996,315.505,-71.603,-176.543,7.774,148.489
C09854=1188.001,315.257,-71.572,-176.545,7.772,148.489
C09855=1188.005,315.008,-71.541,-176.547,7.769,148.489
C09856=1188.009,314.733,-71.506,-176.551,7.765,148.489
C09857=1188.013,314.456,-71.472,-176.553,7.762,148.489
C09858=1188.019,314.179,-71.438,-176.556,7.759,148.489
C09859=1188.023,313.903,-71.403,-176.558,7.756,148.489
C09860=1188.028,313.655,-71.372,-176.561,7.753,148.489
C09861=1188.032,313.406,-71.341,-176.564,7.750,148.489
C09862=1188.036,313.159,-71.311,-176.566,7.747,148.489
C09863=1188.041,312.911,-71.280,-176.569,7.743,148.489
C09864=1188.045,312.662,-71.249,-176.571,7.740,148.489
C09865=1188.049,312.414,-71.218,-176.573,7.738,148.489
C09866=1188.053,312.167,-71.187,-176.576,7.735,148.489
C09867=1188.057,311.918,-71.156,-176.578,7.732,148.489
C09868=1188.061,311.670,-71.125,-176.581,7.729,148.489
C09869=1188.066,311.422,-71.095,-176.584,7.726,148.489
C09870=1188.070,311.175,-71.064,-176.585,7.723,148.489
C09871=1188.074,310.926,-71.033,-176.588,7.720,148.489
C09872=1188.079,310.677,-71.003,-176.591,7.717,148.489
C09873=1188.083,310.430,-70.973,-176.594,7.714,148.489
C09874=1188.087,310.182,-70.942,-176.596,7.711,148.488
C09875=1188.091,309.933,-70.911,-176.599,7.708,148.488
C09876=1188.095,309.686,-70.881,-176.601,7.706,148.489
C09877=1188.100,309.438,-70.850,-176.603,7.703,148.489
C09878=1188.104,309.190,-70.820,-176.606,7.700,148.488
C09879=1188.108,308.941,-70.789,-176.608,7.697,148.488
C09880=1188.112,308.693,-70.758,-176.611,7.694,148.488
C09881=1188.117,308.445,-70.729,-176.613,7.691,148.488
C09882=1188.121,308.197,-70.698,-176.615,7.688,148.488
C09883=1188.125,307.948,-70.667,-176.618,7.685,148.488
C09884=1188.129,307.701,-70.637,-176.621,7.682,148.488
C09885=1188.134,307.453,-70.606,-176.624,7.679,148.488
C09886=1188.138,307.205,-70.576,-176.626,7.676,148.488
C09887=1188.142,306.957,-70.546,-176.628,7.674,148.488
C09888=1188.146,306.708,-70.515,-176.631,7.671,148.488
C09889=1188.150,306.460,-70.484,-176.633,7.668,148.488
C09890=1188.155,306.212,-70.454,-176.636,7.665,148.488
C09891=1188.159,305.964,-70.424,-176.639,7.662,148.488
C09892=1188.164,305.716,-70.393,-176.641,7.659,148.488
C09893=1188.168,305.469,-70.363,-176.643,7.656,148.488
C09894=1188.172,305.219,-70.333,-176.646,7.653,148.488
C09895=1188.176,304.972,-70.303,-176.649,7.650,148.488
C09896=1188.180,304.724,-70.272,-176.651,7.647,148.488
C09897=1188.185,304.475,-70.242,-176.653,7.645,148.488
C09898=1188.189,304.227,-70.212,-176.656,7.642,148.488
C09899=1188.193,303.979,-70.182,-176.658,7.639,148.488
C09900=1188.198,303.731,-70.151,-176.661,7.636,148.488
C09901=1188.201,303.483,-70.121,-176.664,7.633,148.488
C09902=1188.206,303.234,-70.091,-176.666,7.630,148.488
C09903=1188.210,302.987,-70.061,-176.668,7.627,148.488
C09904=1188.215,302.738,-70.031,-176.671,7.624,148.488
C09905=1188.219,302.490,-70.001,-176.674,7.621,148.488
C09906=1188.223,302.242,-69.971,-176.676,7.619,148.488
C09907=1188.228,301.994,-69.940,-176.679,7.616,148.488
C09908=1188.232,301.746,-69.911,-176.681,7.613,148.488
C09909=1188.236,301.498,-69.880,-176.684,7.610,148.488
C09910=1188.241,301.250,-69.851,-176.686,7.607,148.488
C09911=1188.244,301.001,-69.820,-176.688,7.604,148.488
C09912=1188.249,300.753,-69.790,-176.691,7.601,148.488
C09913=1188.253,300.505,-69.760,-176.694,7.598,148.488
C09914=1188.257,300.257,-69.730,-176.697,7.595,148.488
C09915=1188.262,300.008,-69.700,-176.699,7.593,148.488
C09916=1188.266,299.761,-69.670,-176.701,7.590,148.488
C09917=1188.270,299.512,-69.641,-176.704,7.587,148.488
C09918=1188.274,299.264,-69.610,-176.706,7.584,148.488
C09919=1188.279,299.016,-69.581,-176.709,7.581,148.488
C09920=1188.283,298.768,-69.551,-176.711,7.579,148.488
C09921=1188.287,298.520,-69.520,-176.714,7.576,148.488
C09922=1188.292,298.272,-69.491,-176.717,7.573,148.488
C09923=1188.296,298.023,-69.461,-176.719,7.570,148.488
C09924=1188.300,297.775,-69.432,-176.722,7.567,148.488
C09925=1188.305,297.527,-69.401,-176.724,7.564,148.488
C09926=1188.309,297.279,-69.372,-176.727,7.561,148.488
C09927=1188.313,297.031,-69.342,-176.730,7.558,148.488
C09928=1188.317,296.782,-69.313,-176.731,7.556,148.488
C09929=1188.322,296.534,-69.282,-176.734,7.553,148.488
C09930=1188.326,296.286,-69.253,-176.737,7.550,148.488
C09931=1188.330,296.038,-69.223,-176.739,7.547,148.488
C09932=1188.334,295.790,-69.194,-176.742,7.545,148.488
C09933=1188.338,295.542,-69.164,-176.744,7.542,148.488
C09934=1188.342,295.294,-69.134,-176.747,7.539,148.488
C09935=1188.347,295.045,-69.104,-176.750,7.536,148.488
C09936=1188.351,294.797,-69.075,-176.752,7.534,148.488
C09937=1188.356,294.549,-69.045,-176.755,7.531,148.488
C09938=1188.360,294.300,-69.016,-176.757,7.528,148.488
C09939=1188.364,294.052,-68.986,-176.760,7.525,148.488
C09940=1188.368,293.804,-68.957,-176.762,7.522,148.488
C09941=1188.372,293.555,-68.927,-176.765,7.519,148.489
C09942=1188.377,293.307,-68.897,-176.768,7.516,148.489
C09943=1188.381,293.059,-68.867,-176.770,7.513,148.489
C09944=1188.385,292.811,-68.838,-176.773,7.511,148.489
C09945=1188.390,292.563,-68.809,-176.775,7.508,148.488
C09946=1188.394,292.315,-68.779,-176.777,7.505,148.488
C09947=1188.398,292.067,-68.750,-176.780,7.502,148.489
C09948=1188.403,291.819,-68.720,-176.782,7.500,148.489
C09949=1188.407,291.570,-68.691,-176.785,7.497,148.489
C09950=1188.411,291.322,-68.661,-176.788,7.494,148.489
C09951=1188.416,291.073,-68.633,-176.791,7.491,148.489
C09952=1188.420,290.825,-68.603,-176.793,7.489,148.489
C09953=1188.424,290.577,-68.574,-176.795,7.486,148.489
C09954=1188.429,290.329,-68.545,-176.798,7.483,148.489
C09955=1188.433,290.081,-68.515,-176.800,7.480,148.489
C09956=1188.437,289.833,-68.486,-176.803,7.477,148.489
C09957=1188.441,289.584,-68.456,-176.806,7.474,148.489
C09958=1188.445,289.336,-68.427,-176.808,7.471,148.489
C09959=1188.450,289.088,-68.397,-176.811,7.469,148.489
C09960=1188.455,288.813,-68.365,-176.813,7.466,148.489
C09961=1188.459,288.538,-68.333,-176.817,7.462,148.489
C09962=1188.464,288.264,-68.301,-176.820,7.460,148.489
C09963=1188.469,287.990,-68.268,-176.822,7.457,148.489
C09964=1188.474,287.741,-68.239,-176.825,7.455,148.489
C09965=1188.478,287.493,-68.210,-176.827,7.452,148.489
C09966=1188.482,287.244,-68.181,-176.830,7.449,148.489
C09967=1188.486,286.996,-68.151,-176.833,7.446,148.489
C09968=1188.490,286.749,-68.123,-176.835,7.443,148.490
C09969=1188.495,286.500,-68.093,-176.838,7.440,148.490
C09970=1188.499,286.251,-68.065,-176.840,7.437,148.490
C09971=1188.503,286.003,-68.035,-176.842,7.435,148.490
C09972=1188.508,285.756,-68.006,-176.845,7.432,148.490
C09973=1188.513,285.507,-67.977,-176.848,7.429,148.490
C09974=1188.517,285.258,-67.948,-176.850,7.427,148.490
C09975=1188.520,285.011,-67.919,-176.853,7.424,148.490
C09976=1188.525,284.762,-67.890,-176.855,7.421,148.490
C09977=1188.529,284.514,-67.861,-176.858,7.418,148.490
C09978=1188.534,284.265,-67.833,-176.860,7.416,148.490
C09979=1188.538,284.017,-67.803,-176.863,7.413,148.490
C09980=1188.543,283.769,-67.774,-176.866,7.410,148.490
C09981=1188.547,283.521,-67.746,-176.868,7.408,148.490
C09982=1188.551,283.272,-67.716,-176.871,7.405,148.490
C09983=1188.555,283.024,-67.688,-176.873,7.402,148.490
C09984=1188.560,282.776,-67.659,-176.876,7.400,148.490
C09985=1188.564,282.527,-67.630,-176.879,7.397,148.491
C09986=1188.568,282.279,-67.601,-176.881,7.394,148.491
C09987=1188.573,282.031,-67.573,-176.884,7.392,148.491
C09988=1188.577,281.783,-67.543,-176.886,7.389,148.491
C09989=1188.581,281.534,-67.515,-176.889,7.386,148.491
C09990=1188.586,281.287,-67.486,-176.891,7.384,148.491
C09991=1188.590,281.038,-67.457,-176.894,7.381,148.491
C09992=1188.595,280.789,-67.428,-176.897,7.378,148.491
C09993=1188.598,280.541,-67.400,-176.899,7.375,148.491
C09994=1188.603,280.293,-67.371,-176.901,7.372,148.491
C09995=1188.608,280.044,-67.342,-176.904,7.369,148.491
C09996=1188.611,279.796,-67.314,-176.906,7.367,148.491
//INST
///DATE 2021/06/25 14:28
///ATTR SC,RW,RJ
////FRAME ROBOT
///GROUP1 RB1
NOP
MOVL C00000 V=800.0 PL=0
MOVL C00001 V=800.0 PL=0
MOVL C00002 V=800.0 PL=0
MOVL C00003 V=800.0 PL=0
MOVL C00004 V=800.0 PL=0
MOVL C00005 V=800.0 PL=0
MOVL C00006 V=800.0 PL=0
MOVL C00007 V=800.0 PL=0
MOVL C00008 V=800.0 PL=0
MOVL C00009 V=800.0 PL=0
MOVL C00010 V=800.0 PL=0
MOVL C00011 V=800.0 PL=0
MOVL C00012 V=800.0 PL=0
MOVL C00013 V=800.0 PL=0
MOVL C00014 V=800.0 PL=0
MOVL C00015 V=800.0 PL=0
MOVL C00016 V=800.0 PL=0
MOVL C00017 V=800.0 PL=0
MOVL C00018 V=800.0 PL=0
MOVL C00019 V=800.0 PL=0
MOVL C00020 V=800.0 PL=0
MOVL C00021 V=800.0 PL=0
MOVL C00022 V=800.0 PL=0
MOVL C00023 V=800.0 PL=0
MOVL C00024 V=800.0 PL=0
MOVL C00025 V=800.0 PL=0
MOVL C00026 V=800.0 PL=0
MOVL C00027 V=800.0 PL=0
MOVL C00028 V=800.0 PL=0
MOVL C00029 V=800.0 PL=0
MOVL C00030 V=800.0 PL=0
MOVL C00031 V=800.0 PL=0
MOVL C00032 V=800.0 PL=0
MOVL C00033 V=800.0 PL=0
MOVL C00034 V=800.0 PL=0
MOVL C00035 V=800.0 PL=0
MOVL C00036 V=800.0 PL=0
MOVL C00037 V=800.0 PL=0
MOVL C00038 V=800.0 PL=0
MOVL C00039 V=800.0 PL=0
MOVL C00040 V=800.0 PL=0
MOVL C00041 V=800.0 PL=0
MOVL C00042 V=800.0 PL=0
MOVL C00043 V=800.0 PL=0
MOVL C00044 V=800.0 PL=0
MOVL C00045 V=800.0 PL=0
MOVL C00046 V=800.0 PL=0
MOVL C00047 V=800.0 PL=0
MOVL C00048 V=800.0 PL=0
MOVL C00049 V=800.0 PL=0
MOVL C00050 V=800.0 PL=0
MOVL C00051 V=800.0 PL=0
MOVL C00052 V=800.0 PL=0
MOVL C00053 V=800.0 PL=0
MOVL C00054 V=800.0 PL=0
MOVL C00055 V=800.0 PL=0
MOVL C00056 V=800.0 PL=0
MOVL C00057 V=800.0 PL=0
MOVL C00058 V=800.0 PL=0
MOVL C00059 V=800.0 PL=0
MOVL C00060 V=800.0 PL=0
MOVL C00061 V=800.0 PL=0
MOVL C00062 V=800.0 PL=0
MOVL C00063 V=800.0 PL=0
MOVL C00064 V=800.0 PL=0
MOVL C00065 V=800.0 PL=0
MOVL C00066 V=800.0 PL=0
MOVL C00067 V=800.0 PL=0
MOVL C00068 V=800.0 PL=0
MOVL C00069 V=800.0 PL=0
MOVL C00070 V=800.0 PL=0
MOVL C00071 V=800.0 PL=0
MOVL C00072 V=800.0 PL=0
MOVL C00073 V=800.0 PL=0
MOVL C00074 V=800.0 PL=0
MOVL C00075 V=800.0 PL=0
MOVL C00076 V=800.0 PL=0
MOVL C00077 V=800.0 PL=0
MOVL C00078 V=800.0 PL=0
MOVL C00079 V=800.0 PL=0
MOVL C00080 V=800.0 PL=0
MOVL C00081 V=800.0 PL=0
MOVL C00082 V=800.0 PL=0
MOVL C00083 V=800.0 PL=0
MOVL C00084 V=800.0 PL=0
MOVL C00085 V=800.0 PL=0
MOVL C00086 V=800.0 PL=0
MOVL C00087 V=800.0 PL=0
MOVL C00088 V=800.0 PL=0
MOVL C00089 V=800.0 PL=0
MOVL C00090 V=800.0 PL=0
MOVL C00091 V=800.0 PL=0
MOVL C00092 V=800.0 PL=0
MOVL C00093 V=800.0 PL=0
MOVL C00094 V=800.0 PL=0
MOVL C00095 V=800.0 PL=0
MOVL C00096 V=800.0 PL=0
MOVL C00097 V=800.0 PL=0
MOVL C00098 V=800.0 PL=0
MOVL C00099 V=800.0 PL=0
MOVL C00100 V=800.0 PL=0
MOVL C00101 V=800.0 PL=0
MOVL C00102 V=800.0 PL=0
MOVL C00103 V=800.0 PL=0
MOVL C00104 V=800.0 PL=0
MOVL C00105 V=800.0 PL=0
MOVL C00106 V=800.0 PL=0
MOVL C00107 V=800.0 PL=0
MOVL C00108 V=800.0 PL=0
MOVL C00109 V=800.0 PL=0
MOVL C00110 V=800.0 PL=0
MOVL C00111 V=800.0 PL=0
MOVL C00112 V=800.0 PL=0
MOVL C00113 V=800.0 PL=0
MOVL C00114 V=800.0 PL=0
MOVL C00115 V=800.0 PL=0
MOVL C00116 V=800.0 PL=0
MOVL C00117 V=800.0 PL=0
MOVL C00118 V=800.0 PL=0
MOVL C00119 V=800.0 PL=0
MOVL C00120 V=800.0 PL=0
MOVL C00121 V=800.0 PL=0
MOVL C00122 V=800.0 PL=0
MOVL C00123 V=800.0 PL=0
MOVL C00124 V=800.0 PL=0
MOVL C00125 V=800.0 PL=0
MOVL C00126 V=800.0 PL=0
MOVL C00127 V=800.0 PL=0
MOVL C00128 V=800.0 PL=0
MOVL C00129 V=800.0 PL=0
MOVL C00130 V=800.0 PL=0
MOVL C00131 V=800.0 PL=0
MOVL C00132 V=800.0 PL=0
MOVL C00133 V=800.0 PL=0
MOVL C00134 V=800.0 PL=0
MOVL C00135 V=800.0 PL=0
MOVL C00136 V=800.0 PL=0
MOVL C00137 V=800.0 PL=0
MOVL C00138 V=800.0 PL=0
MOVL C00139 V=800.0 PL=0
MOVL C00140 V=800.0 PL=0
MOVL C00141 V=800.0 PL=0
MOVL C00142 V=800.0 PL=0
MOVL C00143 V=800.0 PL=0
MOVL C00144 V=800.0 PL=0
MOVL C00145 V=800.0 PL=0
MOVL C00146 V=800.0 PL=0
MOVL C00147 V=800.0 PL=0
MOVL C00148 V=800.0 PL=0
MOVL C00149 V=800.0 PL=0
MOVL C00150 V=800.0 PL=0
MOVL C00151 V=800.0 PL=0
MOVL C00152 V=800.0 PL=0
MOVL C00153 V=800.0 PL=0
MOVL C00154 V=800.0 PL=0
MOVL C00155 V=800.0 PL=0
MOVL C00156 V=800.0 PL=0
MOVL C00157 V=800.0 PL=0
MOVL C00158 V=800.0 PL=0
MOVL C00159 V=800.0 PL=0
MOVL C00160 V=800.0 PL=0
MOVL C00161 V=800.0 PL=0
MOVL C00162 V=800.0 PL=0
MOVL C00163 V=800.0 PL=0
MOVL C00164 V=800.0 PL=0
MOVL C00165 V=800.0 PL=0
MOVL C00166 V=800.0 PL=0
MOVL C00167 V=800.0 PL=0
MOVL C00168 V=800.0 PL=0
MOVL C00169 V=800.0 PL=0
MOVL C00170 V=800.0 PL=0
MOVL C00171 V=800.0 PL=0
MOVL C00172 V=800.0 PL=0
MOVL C00173 V=800.0 PL=0
MOVL C00174 V=800.0 PL=0
MOVL C00175 V=800.0 PL=0
MOVL C00176 V=800.0 PL=0
MOVL C00177 V=800.0 PL=0
MOVL C00178 V=800.0 PL=0
MOVL C00179 V=800.0 PL=0
MOVL C00180 V=800.0 PL=0
MOVL C00181 V=800.0 PL=0
MOVL C00182 V=800.0 PL=0
MOVL C00183 V=800.0 PL=0
MOVL C00184 V=800.0 PL=0
MOVL C00185 V=800.0 PL=0
MOVL C00186 V=800.0 PL=0
MOVL C00187 V=800.0 PL=0
MOVL C00188 V=800.0 PL=0
MOVL C00189 V=800.0 PL=0
MOVL C00190 V=800.0 PL=0
MOVL C00191 V=800.0 PL=0
MOVL C00192 V=800.0 PL=0
MOVL C00193 V=800.0 PL=0
MOVL C00194 V=800.0 PL=0
MOVL C00195 V=800.0 PL=0
MOVL C00196 V=800.0 PL=0
MOVL C00197 V=800.0 PL=0
MOVL C00198 V=800.0 PL=0
MOVL C00199 V=800.0 PL=0
MOVL C00200 V=800.0 PL=0
MOVL C00201 V=800.0 PL=0
MOVL C00202 V=800.0 PL=0
MOVL C00203 V=800.0 PL=0
MOVL C00204 V=800.0 PL=0
MOVL C00205 V=800.0 PL=0
MOVL C00206 V=800.0 PL=0
MOVL C00207 V=800.0 PL=0
MOVL C00208 V=800.0 PL=0
MOVL C00209 V=800.0 PL=0
MOVL C00210 V=800.0 PL=0
MOVL C00211 V=800.0 PL=0
MOVL C00212 V=800.0 PL=0
MOVL C00213 V=800.0 PL=0
MOVL C00214 V=800.0 PL=0
MOVL C00215 V=800.0 PL=0
MOVL C00216 V=800.0 PL=0
MOVL C00217 V=800.0 PL=0
MOVL C00218 V=800.0 PL=0
MOVL C00219 V=800.0 PL=0
MOVL C00220 V=800.0 PL=0
MOVL C00221 V=800.0 PL=0
MOVL C00222 V=800.0 PL=0
MOVL C00223 V=800.0 PL=0
MOVL C00224 V=800.0 PL=0
MOVL C00225 V=800.0 PL=0
MOVL C00226 V=800.0 PL=0
MOVL C00227 V=800.0 PL=0
MOVL C00228 V=800.0 PL=0
MOVL C00229 V=800.0 PL=0
MOVL C00230 V=800.0 PL=0
MOVL C00231 V=800.0 PL=0
MOVL C00232 V=800.0 PL=0
MOVL C00233 V=800.0 PL=0
MOVL C00234 V=800.0 PL=0
MOVL C00235 V=800.0 PL=0
MOVL C00236 V=800.0 PL=0
MOVL C00237 V=800.0 PL=0
MOVL C00238 V=800.0 PL=0
MOVL C00239 V=800.0 PL=0
MOVL C00240 V=800.0 PL=0
MOVL C00241 V=800.0 PL=0
MOVL C00242 V=800.0 PL=0
MOVL C00243 V=800.0 PL=0
MOVL C00244 V=800.0 PL=0
MOVL C00245 V=800.0 PL=0
MOVL C00246 V=800.0 PL=0
MOVL C00247 V=800.0 PL=0
MOVL C00248 V=800.0 PL=0
MOVL C00249 V=800.0 PL=0
MOVL C00250 V=800.0 PL=0
MOVL C00251 V=800.0 PL=0
MOVL C00252 V=800.0 PL=0
MOVL C00253 V=800.0 PL=0
MOVL C00254 V=800.0 PL=0
MOVL C00255 V=800.0 PL=0
MOVL C00256 V=800.0 PL=0
MOVL C00257 V=800.0 PL=0
MOVL C00258 V=800.0 PL=0
MOVL C00259 V=800.0 PL=0
MOVL C00260 V=800.0 PL=0
MOVL C00261 V=800.0 PL=0
MOVL C00262 V=800.0 PL=0
MOVL C00263 V=800.0 PL=0
MOVL C00264 V=800.0 PL=0
MOVL C00265 V=800.0 PL=0
MOVL C00266 V=800.0 PL=0
MOVL C00267 V=800.0 PL=0
MOVL C00268 V=800.0 PL=0
MOVL C00269 V=800.0 PL=0
MOVL C00270 V=800.0 PL=0
MOVL C00271 V=800.0 PL=0
MOVL C00272 V=800.0 PL=0
MOVL C00273 V=800.0 PL=0
MOVL C00274 V=800.0 PL=0
MOVL C00275 V=800.0 PL=0
MOVL C00276 V=800.0 PL=0
MOVL C00277 V=800.0 PL=0
MOVL C00278 V=800.0 PL=0
MOVL C00279 V=800.0 PL=0
MOVL C00280 V=800.0 PL=0
MOVL C00281 V=800.0 PL=0
MOVL C00282 V=800.0 PL=0
MOVL C00283 V=800.0 PL=0
MOVL C00284 V=800.0 PL=0
MOVL C00285 V=800.0 PL=0
MOVL C00286 V=800.0 PL=0
MOVL C00287 V=800.0 PL=0
MOVL C00288 V=800.0 PL=0
MOVL C00289 V=800.0 PL=0
MOVL C00290 V=800.0 PL=0
MOVL C00291 V=800.0 PL=0
MOVL C00292 V=800.0 PL=0
MOVL C00293 V=800.0 PL=0
MOVL C00294 V=800.0 PL=0
MOVL C00295 V=800.0 PL=0
MOVL C00296 V=800.0 PL=0
MOVL C00297 V=800.0 PL=0
MOVL C00298 V=800.0 PL=0
MOVL C00299 V=800.0 PL=0
MOVL C00300 V=800.0 PL=0
MOVL C00301 V=800.0 PL=0
MOVL C00302 V=800.0 PL=0
MOVL C00303 V=800.0 PL=0
MOVL C00304 V=800.0 PL=0
MOVL C00305 V=800.0 PL=0
MOVL C00306 V=800.0 PL=0
MOVL C00307 V=800.0 PL=0
MOVL C00308 V=800.0 PL=0
MOVL C00309 V=800.0 PL=0
MOVL C00310 V=800.0 PL=0
MOVL C00311 V=800.0 PL=0
MOVL C00312 V=800.0 PL=0
MOVL C00313 V=800.0 PL=0
MOVL C00314 V=800.0 PL=0
MOVL C00315 V=800.0 PL=0
MOVL C00316 V=800.0 PL=0
MOVL C00317 V=800.0 PL=0
MOVL C00318 V=800.0 PL=0
MOVL C00319 V=800.0 PL=0
MOVL C00320 V=800.0 PL=0
MOVL C00321 V=800.0 PL=0
MOVL C00322 V=800.0 PL=0
MOVL C00323 V=800.0 PL=0
MOVL C00324 V=800.0 PL=0
MOVL C00325 V=800.0 PL=0
MOVL C00326 V=800.0 PL=0
MOVL C00327 V=800.0 PL=0
MOVL C00328 V=800.0 PL=0
MOVL C00329 V=800.0 PL=0
MOVL C00330 V=800.0 PL=0
MOVL C00331 V=800.0 PL=0
MOVL C00332 V=800.0 PL=0
MOVL C00333 V=800.0 PL=0
MOVL C00334 V=800.0 PL=0
MOVL C00335 V=800.0 PL=0
MOVL C00336 V=800.0 PL=0
MOVL C00337 V=800.0 PL=0
MOVL C00338 V=800.0 PL=0
MOVL C00339 V=800.0 PL=0
MOVL C00340 V=800.0 PL=0
MOVL C00341 V=800.0 PL=0
MOVL C00342 V=800.0 PL=0
MOVL C00343 V=800.0 PL=0
MOVL C00344 V=800.0 PL=0
MOVL C00345 V=800.0 PL=0
MOVL C00346 V=800.0 PL=0
MOVL C00347 V=800.0 PL=0
MOVL C00348 V=800.0 PL=0
MOVL C00349 V=800.0 PL=0
MOVL C00350 V=800.0 PL=0
MOVL C00351 V=800.0 PL=0
MOVL C00352 V=800.0 PL=0
MOVL C00353 V=800.0 PL=0
MOVL C00354 V=800.0 PL=0
MOVL C00355 V=800.0 PL=0
MOVL C00356 V=800.0 PL=0
MOVL C00357 V=800.0 PL=0
MOVL C00358 V=800.0 PL=0
MOVL C00359 V=800.0 PL=0
MOVL C00360 V=800.0 PL=0
MOVL C00361 V=800.0 PL=0
MOVL C00362 V=800.0 PL=0
MOVL C00363 V=800.0 PL=0
MOVL C00364 V=800.0 PL=0
MOVL C00365 V=800.0 PL=0
MOVL C00366 V=800.0 PL=0
MOVL C00367 V=800.0 PL=0
MOVL C00368 V=800.0 PL=0
MOVL C00369 V=800.0 PL=0
MOVL C00370 V=800.0 PL=0
MOVL C00371 V=800.0 PL=0
MOVL C00372 V=800.0 PL=0
MOVL C00373 V=800.0 PL=0
MOVL C00374 V=800.0 PL=0
MOVL C00375 V=800.0 PL=0
MOVL C00376 V=800.0 PL=0
MOVL C00377 V=800.0 PL=0
MOVL C00378 V=800.0 PL=0
MOVL C00379 V=800.0 PL=0
MOVL C00380 V=800.0 PL=0
MOVL C00381 V=800.0 PL=0
MOVL C00382 V=800.0 PL=0
MOVL C00383 V=800.0 PL=0
MOVL C00384 V=800.0 PL=0
MOVL C00385 V=800.0 PL=0
MOVL C00386 V=800.0 PL=0
MOVL C00387 V=800.0 PL=0
MOVL C00388 V=800.0 PL=0
MOVL C00389 V=800.0 PL=0
MOVL C00390 V=800.0 PL=0
MOVL C00391 V=800.0 PL=0
MOVL C00392 V=800.0 PL=0
MOVL C00393 V=800.0 PL=0
MOVL C00394 V=800.0 PL=0
MOVL C00395 V=800.0 PL=0
MOVL C00396 V=800.0 PL=0
MOVL C00397 V=800.0 PL=0
MOVL C00398 V=800.0 PL=0
MOVL C00399 V=800.0 PL=0
MOVL C00400 V=800.0 PL=0
MOVL C00401 V=800.0 PL=0
MOVL C00402 V=800.0 PL=0
MOVL C00403 V=800.0 PL=0
MOVL C00404 V=800.0 PL=0
MOVL C00405 V=800.0 PL=0
MOVL C00406 V=800.0 PL=0
MOVL C00407 V=800.0 PL=0
MOVL C00408 V=800.0 PL=0
MOVL C00409 V=800.0 PL=0
MOVL C00410 V=800.0 PL=0
MOVL C00411 V=800.0 PL=0
MOVL C00412 V=800.0 PL=0
MOVL C00413 V=800.0 PL=0
MOVL C00414 V=800.0 PL=0
MOVL C00415 V=800.0 PL=0
MOVL C00416 V=800.0 PL=0
MOVL C00417 V=800.0 PL=0
MOVL C00418 V=800.0 PL=0
MOVL C00419 V=800.0 PL=0
MOVL C00420 V=800.0 PL=0
MOVL C00421 V=800.0 PL=0
MOVL C00422 V=800.0 PL=0
MOVL C00423 V=800.0 PL=0
MOVL C00424 V=800.0 PL=0
MOVL C00425 V=800.0 PL=0
MOVL C00426 V=800.0 PL=0
MOVL C00427 V=800.0 PL=0
MOVL C00428 V=800.0 PL=0
MOVL C00429 V=800.0 PL=0
MOVL C00430 V=800.0 PL=0
MOVL C00431 V=800.0 PL=0
MOVL C00432 V=800.0 PL=0
MOVL C00433 V=800.0 PL=0
MOVL C00434 V=800.0 PL=0
MOVL C00435 V=800.0 PL=0
MOVL C00436 V=800.0 PL=0
MOVL C00437 V=800.0 PL=0
MOVL C00438 V=800.0 PL=0
MOVL C00439 V=800.0 PL=0
MOVL C00440 V=800.0 PL=0
MOVL C00441 V=800.0 PL=0
MOVL C00442 V=800.0 PL=0
MOVL C00443 V=800.0 PL=0
MOVL C00444 V=800.0 PL=0
MOVL C00445 V=800.0 PL=0
MOVL C00446 V=800.0 PL=0
MOVL C00447 V=800.0 PL=0
MOVL C00448 V=800.0 PL=0
MOVL C00449 V=800.0 PL=0
MOVL C00450 V=800.0 PL=0
MOVL C00451 V=800.0 PL=0
MOVL C00452 V=800.0 PL=0
MOVL C00453 V=800.0 PL=0
MOVL C00454 V=800.0 PL=0
MOVL C00455 V=800.0 PL=0
MOVL C00456 V=800.0 PL=0
MOVL C00457 V=800.0 PL=0
MOVL C00458 V=800.0 PL=0
MOVL C00459 V=800.0 PL=0
MOVL C00460 V=800.0 PL=0
MOVL C00461 V=800.0 PL=0
MOVL C00462 V=800.0 PL=0
MOVL C00463 V=800.0 PL=0
MOVL C00464 V=800.0 PL=0
MOVL C00465 V=800.0 PL=0
MOVL C00466 V=800.0 PL=0
MOVL C00467 V=800.0 PL=0
MOVL C00468 V=800.0 PL=0
MOVL C00469 V=800.0 PL=0
MOVL C00470 V=800.0 PL=0
MOVL C00471 V=800.0 PL=0
MOVL C00472 V=800.0 PL=0
MOVL C00473 V=800.0 PL=0
MOVL C00474 V=800.0 PL=0
MOVL C00475 V=800.0 PL=0
MOVL C00476 V=800.0 PL=0
MOVL C00477 V=800.0 PL=0
MOVL C00478 V=800.0 PL=0
MOVL C00479 V=800.0 PL=0
MOVL C00480 V=800.0 PL=0
MOVL C00481 V=800.0 PL=0
MOVL C00482 V=800.0 PL=0
MOVL C00483 V=800.0 PL=0
MOVL C00484 V=800.0 PL=0
MOVL C00485 V=800.0 PL=0
MOVL C00486 V=800.0 PL=0
MOVL C00487 V=800.0 PL=0
MOVL C00488 V=800.0 PL=0
MOVL C00489 V=800.0 PL=0
MOVL C00490 V=800.0 PL=0
MOVL C00491 V=800.0 PL=0
MOVL C00492 V=800.0 PL=0
MOVL C00493 V=800.0 PL=0
MOVL C00494 V=800.0 PL=0
MOVL C00495 V=800.0 PL=0
MOVL C00496 V=800.0 PL=0
MOVL C00497 V=800.0 PL=0
MOVL C00498 V=800.0 PL=0
MOVL C00499 V=800.0 PL=0
MOVL C00500 V=800.0 PL=0
MOVL C00501 V=800.0 PL=0
MOVL C00502 V=800.0 PL=0
MOVL C00503 V=800.0 PL=0
MOVL C00504 V=800.0 PL=0
MOVL C00505 V=800.0 PL=0
MOVL C00506 V=800.0 PL=0
MOVL C00507 V=800.0 PL=0
MOVL C00508 V=800.0 PL=0
MOVL C00509 V=800.0 PL=0
MOVL C00510 V=800.0 PL=0
MOVL C00511 V=800.0 PL=0
MOVL C00512 V=800.0 PL=0
MOVL C00513 V=800.0 PL=0
MOVL C00514 V=800.0 PL=0
MOVL C00515 V=800.0 PL=0
MOVL C00516 V=800.0 PL=0
MOVL C00517 V=800.0 PL=0
MOVL C00518 V=800.0 PL=0
MOVL C00519 V=800.0 PL=0
MOVL C00520 V=800.0 PL=0
MOVL C00521 V=800.0 PL=0
MOVL C00522 V=800.0 PL=0
MOVL C00523 V=800.0 PL=0
MOVL C00524 V=800.0 PL=0
MOVL C00525 V=800.0 PL=0
MOVL C00526 V=800.0 PL=0
MOVL C00527 V=800.0 PL=0
MOVL C00528 V=800.0 PL=0
MOVL C00529 V=800.0 PL=0
MOVL C00530 V=800.0 PL=0
MOVL C00531 V=800.0 PL=0
MOVL C00532 V=800.0 PL=0
MOVL C00533 V=800.0 PL=0
MOVL C00534 V=800.0 PL=0
MOVL C00535 V=800.0 PL=0
MOVL C00536 V=800.0 PL=0
MOVL C00537 V=800.0 PL=0
MOVL C00538 V=800.0 PL=0
MOVL C00539 V=800.0 PL=0
MOVL C00540 V=800.0 PL=0
MOVL C00541 V=800.0 PL=0
MOVL C00542 V=800.0 PL=0
MOVL C00543 V=800.0 PL=0
MOVL C00544 V=800.0 PL=0
MOVL C00545 V=800.0 PL=0
MOVL C00546 V=800.0 PL=0
MOVL C00547 V=800.0 PL=0
MOVL C00548 V=800.0 PL=0
MOVL C00549 V=800.0 PL=0
MOVL C00550 V=800.0 PL=0
MOVL C00551 V=800.0 PL=0
MOVL C00552 V=800.0 PL=0
MOVL C00553 V=800.0 PL=0
MOVL C00554 V=800.0 PL=0
MOVL C00555 V=800.0 PL=0
MOVL C00556 V=800.0 PL=0
MOVL C00557 V=800.0 PL=0
MOVL C00558 V=800.0 PL=0
MOVL C00559 V=800.0 PL=0
MOVL C00560 V=800.0 PL=0
MOVL C00561 V=800.0 PL=0
MOVL C00562 V=800.0 PL=0
MOVL C00563 V=800.0 PL=0
MOVL C00564 V=800.0 PL=0
MOVL C00565 V=800.0 PL=0
MOVL C00566 V=800.0 PL=0
MOVL C00567 V=800.0 PL=0
MOVL C00568 V=800.0 PL=0
MOVL C00569 V=800.0 PL=0
MOVL C00570 V=800.0 PL=0
MOVL C00571 V=800.0 PL=0
MOVL C00572 V=800.0 PL=0
MOVL C00573 V=800.0 PL=0
MOVL C00574 V=800.0 PL=0
MOVL C00575 V=800.0 PL=0
MOVL C00576 V=800.0 PL=0
MOVL C00577 V=800.0 PL=0
MOVL C00578 V=800.0 PL=0
MOVL C00579 V=800.0 PL=0
MOVL C00580 V=800.0 PL=0
MOVL C00581 V=800.0 PL=0
MOVL C00582 V=800.0 PL=0
MOVL C00583 V=800.0 PL=0
MOVL C00584 V=800.0 PL=0
MOVL C00585 V=800.0 PL=0
MOVL C00586 V=800.0 PL=0
MOVL C00587 V=800.0 PL=0
MOVL C00588 V=800.0 PL=0
MOVL C00589 V=800.0 PL=0
MOVL C00590 V=800.0 PL=0
MOVL C00591 V=800.0 PL=0
MOVL C00592 V=800.0 PL=0
MOVL C00593 V=800.0 PL=0
MOVL C00594 V=800.0 PL=0
MOVL C00595 V=800.0 PL=0
MOVL C00596 V=800.0 PL=0
MOVL C00597 V=800.0 PL=0
MOVL C00598 V=800.0 PL=0
MOVL C00599 V=800.0 PL=0
MOVL C00600 V=800.0 PL=0
MOVL C00601 V=800.0 PL=0
MOVL C00602 V=800.0 PL=0
MOVL C00603 V=800.0 PL=0
MOVL C00604 V=800.0 PL=0
MOVL C00605 V=800.0 PL=0
MOVL C00606 V=800.0 PL=0
MOVL C00607 V=800.0 PL=0
MOVL C00608 V=800.0 PL=0
MOVL C00609 V=800.0 PL=0
MOVL C00610 V=800.0 PL=0
MOVL C00611 V=800.0 PL=0
MOVL C00612 V=800.0 PL=0
MOVL C00613 V=800.0 PL=0
MOVL C00614 V=800.0 PL=0
MOVL C00615 V=800.0 PL=0
MOVL C00616 V=800.0 PL=0
MOVL C00617 V=800.0 PL=0
MOVL C00618 V=800.0 PL=0
MOVL C00619 V=800.0 PL=0
MOVL C00620 V=800.0 PL=0
MOVL C00621 V=800.0 PL=0
MOVL C00622 V=800.0 PL=0
MOVL C00623 V=800.0 PL=0
MOVL C00624 V=800.0 PL=0
MOVL C00625 V=800.0 PL=0
MOVL C00626 V=800.0 PL=0
MOVL C00627 V=800.0 PL=0
MOVL C00628 V=800.0 PL=0
MOVL C00629 V=800.0 PL=0
MOVL C00630 V=800.0 PL=0
MOVL C00631 V=800.0 PL=0
MOVL C00632 V=800.0 PL=0
MOVL C00633 V=800.0 PL=0
MOVL C00634 V=800.0 PL=0
MOVL C00635 V=800.0 PL=0
MOVL C00636 V=800.0 PL=0
MOVL C00637 V=800.0 PL=0
MOVL C00638 V=800.0 PL=0
MOVL C00639 V=800.0 PL=0
MOVL C00640 V=800.0 PL=0
MOVL C00641 V=800.0 PL=0
MOVL C00642 V=800.0 PL=0
MOVL C00643 V=800.0 PL=0
MOVL C00644 V=800.0 PL=0
MOVL C00645 V=800.0 PL=0
MOVL C00646 V=800.0 PL=0
MOVL C00647 V=800.0 PL=0
MOVL C00648 V=800.0 PL=0
MOVL C00649 V=800.0 PL=0
MOVL C00650 V=800.0 PL=0
MOVL C00651 V=800.0 PL=0
MOVL C00652 V=800.0 PL=0
MOVL C00653 V=800.0 PL=0
MOVL C00654 V=800.0 PL=0
MOVL C00655 V=800.0 PL=0
MOVL C00656 V=800.0 PL=0
MOVL C00657 V=800.0 PL=0
MOVL C00658 V=800.0 PL=0
MOVL C00659 V=800.0 PL=0
MOVL C00660 V=800.0 PL=0
MOVL C00661 V=800.0 PL=0
MOVL C00662 V=800.0 PL=0
MOVL C00663 V=800.0 PL=0
MOVL C00664 V=800.0 PL=0
MOVL C00665 V=800.0 PL=0
MOVL C00666 V=800.0 PL=0
MOVL C00667 V=800.0 PL=0
MOVL C00668 V=800.0 PL=0
MOVL C00669 V=800.0 PL=0
MOVL C00670 V=800.0 PL=0
MOVL C00671 V=800.0 PL=0
MOVL C00672 V=800.0 PL=0
MOVL C00673 V=800.0 PL=0
MOVL C00674 V=800.0 PL=0
MOVL C00675 V=800.0 PL=0
MOVL C00676 V=800.0 PL=0
MOVL C00677 V=800.0 PL=0
MOVL C00678 V=800.0 PL=0
MOVL C00679 V=800.0 PL=0
MOVL C00680 V=800.0 PL=0
MOVL C00681 V=800.0 PL=0
MOVL C00682 V=800.0 PL=0
MOVL C00683 V=800.0 PL=0
MOVL C00684 V=800.0 PL=0
MOVL C00685 V=800.0 PL=0
MOVL C00686 V=800.0 PL=0
MOVL C00687 V=800.0 PL=0
MOVL C00688 V=800.0 PL=0
MOVL C00689 V=800.0 PL=0
MOVL C00690 V=800.0 PL=0
MOVL C00691 V=800.0 PL=0
MOVL C00692 V=800.0 PL=0
MOVL C00693 V=800.0 PL=0
MOVL C00694 V=800.0 PL=0
MOVL C00695 V=800.0 PL=0
MOVL C00696 V=800.0 PL=0
MOVL C00697 V=800.0 PL=0
MOVL C00698 V=800.0 PL=0
MOVL C00699 V=800.0 PL=0
MOVL C00700 V=800.0 PL=0
MOVL C00701 V=800.0 PL=0
MOVL C00702 V=800.0 PL=0
MOVL C00703 V=800.0 PL=0
MOVL C00704 V=800.0 PL=0
MOVL C00705 V=800.0 PL=0
MOVL C00706 V=800.0 PL=0
MOVL C00707 V=800.0 PL=0
MOVL C00708 V=800.0 PL=0
MOVL C00709 V=800.0 PL=0
MOVL C00710 V=800.0 PL=0
MOVL C00711 V=800.0 PL=0
MOVL C00712 V=800.0 PL=0
MOVL C00713 V=800.0 PL=0
MOVL C00714 V=800.0 PL=0
MOVL C00715 V=800.0 PL=0
MOVL C00716 V=800.0 PL=0
MOVL C00717 V=800.0 PL=0
MOVL C00718 V=800.0 PL=0
MOVL C00719 V=800.0 PL=0
MOVL C00720 V=800.0 PL=0
MOVL C00721 V=800.0 PL=0
MOVL C00722 V=800.0 PL=0
MOVL C00723 V=800.0 PL=0
MOVL C00724 V=800.0 PL=0
MOVL C00725 V=800.0 PL=0
MOVL C00726 V=800.0 PL=0
MOVL C00727 V=800.0 PL=0
MOVL C00728 V=800.0 PL=0
MOVL C00729 V=800.0 PL=0
MOVL C00730 V=800.0 PL=0
MOVL C00731 V=800.0 PL=0
MOVL C00732 V=800.0 PL=0
MOVL C00733 V=800.0 PL=0
MOVL C00734 V=800.0 PL=0
MOVL C00735 V=800.0 PL=0
MOVL C00736 V=800.0 PL=0
MOVL C00737 V=800.0 PL=0
MOVL C00738 V=800.0 PL=0
MOVL C00739 V=800.0 PL=0
MOVL C00740 V=800.0 PL=0
MOVL C00741 V=800.0 PL=0
MOVL C00742 V=800.0 PL=0
MOVL C00743 V=800.0 PL=0
MOVL C00744 V=800.0 PL=0
MOVL C00745 V=800.0 PL=0
MOVL C00746 V=800.0 PL=0
MOVL C00747 V=800.0 PL=0
MOVL C00748 V=800.0 PL=0
MOVL C00749 V=800.0 PL=0
MOVL C00750 V=800.0 PL=0
MOVL C00751 V=800.0 PL=0
MOVL C00752 V=800.0 PL=0
MOVL C00753 V=800.0 PL=0
MOVL C00754 V=800.0 PL=0
MOVL C00755 V=800.0 PL=0
MOVL C00756 V=800.0 PL=0
MOVL C00757 V=800.0 PL=0
MOVL C00758 V=800.0 PL=0
MOVL C00759 V=800.0 PL=0
MOVL C00760 V=800.0 PL=0
MOVL C00761 V=800.0 PL=0
MOVL C00762 V=800.0 PL=0
MOVL C00763 V=800.0 PL=0
MOVL C00764 V=800.0 PL=0
MOVL C00765 V=800.0 PL=0
MOVL C00766 V=800.0 PL=0
MOVL C00767 V=800.0 PL=0
MOVL C00768 V=800.0 PL=0
MOVL C00769 V=800.0 PL=0
MOVL C00770 V=800.0 PL=0
MOVL C00771 V=800.0 PL=0
MOVL C00772 V=800.0 PL=0
MOVL C00773 V=800.0 PL=0
MOVL C00774 V=800.0 PL=0
MOVL C00775 V=800.0 PL=0
MOVL C00776 V=800.0 PL=0
MOVL C00777 V=800.0 PL=0
MOVL C00778 V=800.0 PL=0
MOVL C00779 V=800.0 PL=0
MOVL C00780 V=800.0 PL=0
MOVL C00781 V=800.0 PL=0
MOVL C00782 V=800.0 PL=0
MOVL C00783 V=800.0 PL=0
MOVL C00784 V=800.0 PL=0
MOVL C00785 V=800.0 PL=0
MOVL C00786 V=800.0 PL=0
MOVL C00787 V=800.0 PL=0
MOVL C00788 V=800.0 PL=0
MOVL C00789 V=800.0 PL=0
MOVL C00790 V=800.0 PL=0
MOVL C00791 V=800.0 PL=0
MOVL C00792 V=800.0 PL=0
MOVL C00793 V=800.0 PL=0
MOVL C00794 V=800.0 PL=0
MOVL C00795 V=800.0 PL=0
MOVL C00796 V=800.0 PL=0
MOVL C00797 V=800.0 PL=0
MOVL C00798 V=800.0 PL=0
MOVL C00799 V=800.0 PL=0
MOVL C00800 V=800.0 PL=0
MOVL C00801 V=800.0 PL=0
MOVL C00802 V=800.0 PL=0
MOVL C00803 V=800.0 PL=0
MOVL C00804 V=800.0 PL=0
MOVL C00805 V=800.0 PL=0
MOVL C00806 V=800.0 PL=0
MOVL C00807 V=800.0 PL=0
MOVL C00808 V=800.0 PL=0
MOVL C00809 V=800.0 PL=0
MOVL C00810 V=800.0 PL=0
MOVL C00811 V=800.0 PL=0
MOVL C00812 V=800.0 PL=0
MOVL C00813 V=800.0 PL=0
MOVL C00814 V=800.0 PL=0
MOVL C00815 V=800.0 PL=0
MOVL C00816 V=800.0 PL=0
MOVL C00817 V=800.0 PL=0
MOVL C00818 V=800.0 PL=0
MOVL C00819 V=800.0 PL=0
MOVL C00820 V=800.0 PL=0
MOVL C00821 V=800.0 PL=0
MOVL C00822 V=800.0 PL=0
MOVL C00823 V=800.0 PL=0
MOVL C00824 V=800.0 PL=0
MOVL C00825 V=800.0 PL=0
MOVL C00826 V=800.0 PL=0
MOVL C00827 V=800.0 PL=0
MOVL C00828 V=800.0 PL=0
MOVL C00829 V=800.0 PL=0
MOVL C00830 V=800.0 PL=0
MOVL C00831 V=800.0 PL=0
MOVL C00832 V=800.0 PL=0
MOVL C00833 V=800.0 PL=0
MOVL C00834 V=800.0 PL=0
MOVL C00835 V=800.0 PL=0
MOVL C00836 V=800.0 PL=0
MOVL C00837 V=800.0 PL=0
MOVL C00838 V=800.0 PL=0
MOVL C00839 V=800.0 PL=0
MOVL C00840 V=800.0 PL=0
MOVL C00841 V=800.0 PL=0
MOVL C00842 V=800.0 PL=0
MOVL C00843 V=800.0 PL=0
MOVL C00844 V=800.0 PL=0
MOVL C00845 V=800.0 PL=0
MOVL C00846 V=800.0 PL=0
MOVL C00847 V=800.0 PL=0
MOVL C00848 V=800.0 PL=0
MOVL C00849 V=800.0 PL=0
MOVL C00850 V=800.0 PL=0
MOVL C00851 V=800.0 PL=0
MOVL C00852 V=800.0 PL=0
MOVL C00853 V=800.0 PL=0
MOVL C00854 V=800.0 PL=0
MOVL C00855 V=800.0 PL=0
MOVL C00856 V=800.0 PL=0
MOVL C00857 V=800.0 PL=0
MOVL C00858 V=800.0 PL=0
MOVL C00859 V=800.0 PL=0
MOVL C00860 V=800.0 PL=0
MOVL C00861 V=800.0 PL=0
MOVL C00862 V=800.0 PL=0
MOVL C00863 V=800.0 PL=0
MOVL C00864 V=800.0 PL=0
MOVL C00865 V=800.0 PL=0
MOVL C00866 V=800.0 PL=0
MOVL C00867 V=800.0 PL=0
MOVL C00868 V=800.0 PL=0
MOVL C00869 V=800.0 PL=0
MOVL C00870 V=800.0 PL=0
MOVL C00871 V=800.0 PL=0
MOVL C00872 V=800.0 PL=0
MOVL C00873 V=800.0 PL=0
MOVL C00874 V=800.0 PL=0
MOVL C00875 V=800.0 PL=0
MOVL C00876 V=800.0 PL=0
MOVL C00877 V=800.0 PL=0
MOVL C00878 V=800.0 PL=0
MOVL C00879 V=800.0 PL=0
MOVL C00880 V=800.0 PL=0
MOVL C00881 V=800.0 PL=0
MOVL C00882 V=800.0 PL=0
MOVL C00883 V=800.0 PL=0
MOVL C00884 V=800.0 PL=0
MOVL C00885 V=800.0 PL=0
MOVL C00886 V=800.0 PL=0
MOVL C00887 V=800.0 PL=0
MOVL C00888 V=800.0 PL=0
MOVL C00889 V=800.0 PL=0
MOVL C00890 V=800.0 PL=0
MOVL C00891 V=800.0 PL=0
MOVL C00892 V=800.0 PL=0
MOVL C00893 V=800.0 PL=0
MOVL C00894 V=800.0 PL=0
MOVL C00895 V=800.0 PL=0
MOVL C00896 V=800.0 PL=0
MOVL C00897 V=800.0 PL=0
MOVL C00898 V=800.0 PL=0
MOVL C00899 V=800.0 PL=0
MOVL C00900 V=800.0 PL=0
MOVL C00901 V=800.0 PL=0
MOVL C00902 V=800.0 PL=0
MOVL C00903 V=800.0 PL=0
MOVL C00904 V=800.0 PL=0
MOVL C00905 V=800.0 PL=0
MOVL C00906 V=800.0 PL=0
MOVL C00907 V=800.0 PL=0
MOVL C00908 V=800.0 PL=0
MOVL C00909 V=800.0 PL=0
MOVL C00910 V=800.0 PL=0
MOVL C00911 V=800.0 PL=0
MOVL C00912 V=800.0 PL=0
MOVL C00913 V=800.0 PL=0
MOVL C00914 V=800.0 PL=0
MOVL C00915 V=800.0 PL=0
MOVL C00916 V=800.0 PL=0
MOVL C00917 V=800.0 PL=0
MOVL C00918 V=800.0 PL=0
MOVL C00919 V=800.0 PL=0
MOVL C00920 V=800.0 PL=0
MOVL C00921 V=800.0 PL=0
MOVL C00922 V=800.0 PL=0
MOVL C00923 V=800.0 PL=0
MOVL C00924 V=800.0 PL=0
MOVL C00925 V=800.0 PL=0
MOVL C00926 V=800.0 PL=0
MOVL C00927 V=800.0 PL=0
MOVL C00928 V=800.0 PL=0
MOVL C00929 V=800.0 PL=0
MOVL C00930 V=800.0 PL=0
MOVL C00931 V=800.0 PL=0
MOVL C00932 V=800.0 PL=0
MOVL C00933 V=800.0 PL=0
MOVL C00934 V=800.0 PL=0
MOVL C00935 V=800.0 PL=0
MOVL C00936 V=800.0 PL=0
MOVL C00937 V=800.0 PL=0
MOVL C00938 V=800.0 PL=0
MOVL C00939 V=800.0 PL=0
MOVL C00940 V=800.0 PL=0
MOVL C00941 V=800.0 PL=0
MOVL C00942 V=800.0 PL=0
MOVL C00943 V=800.0 PL=0
MOVL C00944 V=800.0 PL=0
MOVL C00945 V=800.0 PL=0
MOVL C00946 V=800.0 PL=0
MOVL C00947 V=800.0 PL=0
MOVL C00948 V=800.0 PL=0
MOVL C00949 V=800.0 PL=0
MOVL C00950 V=800.0 PL=0
MOVL C00951 V=800.0 PL=0
MOVL C00952 V=800.0 PL=0
MOVL C00953 V=800.0 PL=0
MOVL C00954 V=800.0 PL=0
MOVL C00955 V=800.0 PL=0
MOVL C00956 V=800.0 PL=0
MOVL C00957 V=800.0 PL=0
MOVL C00958 V=800.0 PL=0
MOVL C00959 V=800.0 PL=0
MOVL C00960 V=800.0 PL=0
MOVL C00961 V=800.0 PL=0
MOVL C00962 V=800.0 PL=0
MOVL C00963 V=800.0 PL=0
MOVL C00964 V=800.0 PL=0
MOVL C00965 V=800.0 PL=0
MOVL C00966 V=800.0 PL=0
MOVL C00967 V=800.0 PL=0
MOVL C00968 V=800.0 PL=0
MOVL C00969 V=800.0 PL=0
MOVL C00970 V=800.0 PL=0
MOVL C00971 V=800.0 PL=0
MOVL C00972 V=800.0 PL=0
MOVL C00973 V=800.0 PL=0
MOVL C00974 V=800.0 PL=0
MOVL C00975 V=800.0 PL=0
MOVL C00976 V=800.0 PL=0
MOVL C00977 V=800.0 PL=0
MOVL C00978 V=800.0 PL=0
MOVL C00979 V=800.0 PL=0
MOVL C00980 V=800.0 PL=0
MOVL C00981 V=800.0 PL=0
MOVL C00982 V=800.0 PL=0
MOVL C00983 V=800.0 PL=0
MOVL C00984 V=800.0 PL=0
MOVL C00985 V=800.0 PL=0
MOVL C00986 V=800.0 PL=0
MOVL C00987 V=800.0 PL=0
MOVL C00988 V=800.0 PL=0
MOVL C00989 V=800.0 PL=0
MOVL C00990 V=800.0 PL=0
MOVL C00991 V=800.0 PL=0
MOVL C00992 V=800.0 PL=0
MOVL C00993 V=800.0 PL=0
MOVL C00994 V=800.0 PL=0
MOVL C00995 V=800.0 PL=0
MOVL C00996 V=800.0 PL=0
MOVL C00997 V=800.0 PL=0
MOVL C00998 V=800.0 PL=0
MOVL C00999 V=800.0 PL=0
MOVL C01000 V=800.0 PL=0
MOVL C01001 V=800.0 PL=0
MOVL C01002 V=800.0 PL=0
MOVL C01003 V=800.0 PL=0
MOVL C01004 V=800.0 PL=0
MOVL C01005 V=800.0 PL=0
MOVL C01006 V=800.0 PL=0
MOVL C01007 V=800.0 PL=0
MOVL C01008 V=800.0 PL=0
MOVL C01009 V=800.0 PL=0
MOVL C01010 V=800.0 PL=0
MOVL C01011 V=800.0 PL=0
MOVL C01012 V=800.0 PL=0
MOVL C01013 V=800.0 PL=0
MOVL C01014 V=800.0 PL=0
MOVL C01015 V=800.0 PL=0
MOVL C01016 V=800.0 PL=0
MOVL C01017 V=800.0 PL=0
MOVL C01018 V=800.0 PL=0
MOVL C01019 V=800.0 PL=0
MOVL C01020 V=800.0 PL=0
MOVL C01021 V=800.0 PL=0
MOVL C01022 V=800.0 PL=0
MOVL C01023 V=800.0 PL=0
MOVL C01024 V=800.0 PL=0
MOVL C01025 V=800.0 PL=0
MOVL C01026 V=800.0 PL=0
MOVL C01027 V=800.0 PL=0
MOVL C01028 V=800.0 PL=0
MOVL C01029 V=800.0 PL=0
MOVL C01030 V=800.0 PL=0
MOVL C01031 V=800.0 PL=0
MOVL C01032 V=800.0 PL=0
MOVL C01033 V=800.0 PL=0
MOVL C01034 V=800.0 PL=0
MOVL C01035 V=800.0 PL=0
MOVL C01036 V=800.0 PL=0
MOVL C01037 V=800.0 PL=0
MOVL C01038 V=800.0 PL=0
MOVL C01039 V=800.0 PL=0
MOVL C01040 V=800.0 PL=0
MOVL C01041 V=800.0 PL=0
MOVL C01042 V=800.0 PL=0
MOVL C01043 V=800.0 PL=0
MOVL C01044 V=800.0 PL=0
MOVL C01045 V=800.0 PL=0
MOVL C01046 V=800.0 PL=0
MOVL C01047 V=800.0 PL=0
MOVL C01048 V=800.0 PL=0
MOVL C01049 V=800.0 PL=0
MOVL C01050 V=800.0 PL=0
MOVL C01051 V=800.0 PL=0
MOVL C01052 V=800.0 PL=0
MOVL C01053 V=800.0 PL=0
MOVL C01054 V=800.0 PL=0
MOVL C01055 V=800.0 PL=0
MOVL C01056 V=800.0 PL=0
MOVL C01057 V=800.0 PL=0
MOVL C01058 V=800.0 PL=0
MOVL C01059 V=800.0 PL=0
MOVL C01060 V=800.0 PL=0
MOVL C01061 V=800.0 PL=0
MOVL C01062 V=800.0 PL=0
MOVL C01063 V=800.0 PL=0
MOVL C01064 V=800.0 PL=0
MOVL C01065 V=800.0 PL=0
MOVL C01066 V=800.0 PL=0
MOVL C01067 V=800.0 PL=0
MOVL C01068 V=800.0 PL=0
MOVL C01069 V=800.0 PL=0
MOVL C01070 V=800.0 PL=0
MOVL C01071 V=800.0 PL=0
MOVL C01072 V=800.0 PL=0
MOVL C01073 V=800.0 PL=0
MOVL C01074 V=800.0 PL=0
MOVL C01075 V=800.0 PL=0
MOVL C01076 V=800.0 PL=0
MOVL C01077 V=800.0 PL=0
MOVL C01078 V=800.0 PL=0
MOVL C01079 V=800.0 PL=0
MOVL C01080 V=800.0 PL=0
MOVL C01081 V=800.0 PL=0
MOVL C01082 V=800.0 PL=0
MOVL C01083 V=800.0 PL=0
MOVL C01084 V=800.0 PL=0
MOVL C01085 V=800.0 PL=0
MOVL C01086 V=800.0 PL=0
MOVL C01087 V=800.0 PL=0
MOVL C01088 V=800.0 PL=0
MOVL C01089 V=800.0 PL=0
MOVL C01090 V=800.0 PL=0
MOVL C01091 V=800.0 PL=0
MOVL C01092 V=800.0 PL=0
MOVL C01093 V=800.0 PL=0
MOVL C01094 V=800.0 PL=0
MOVL C01095 V=800.0 PL=0
MOVL C01096 V=800.0 PL=0
MOVL C01097 V=800.0 PL=0
MOVL C01098 V=800.0 PL=0
MOVL C01099 V=800.0 PL=0
MOVL C01100 V=800.0 PL=0
MOVL C01101 V=800.0 PL=0
MOVL C01102 V=800.0 PL=0
MOVL C01103 V=800.0 PL=0
MOVL C01104 V=800.0 PL=0
MOVL C01105 V=800.0 PL=0
MOVL C01106 V=800.0 PL=0
MOVL C01107 V=800.0 PL=0
MOVL C01108 V=800.0 PL=0
MOVL C01109 V=800.0 PL=0
MOVL C01110 V=800.0 PL=0
MOVL C01111 V=800.0 PL=0
MOVL C01112 V=800.0 PL=0
MOVL C01113 V=800.0 PL=0
MOVL C01114 V=800.0 PL=0
MOVL C01115 V=800.0 PL=0
MOVL C01116 V=800.0 PL=0
MOVL C01117 V=800.0 PL=0
MOVL C01118 V=800.0 PL=0
MOVL C01119 V=800.0 PL=0
MOVL C01120 V=800.0 PL=0
MOVL C01121 V=800.0 PL=0
MOVL C01122 V=800.0 PL=0
MOVL C01123 V=800.0 PL=0
MOVL C01124 V=800.0 PL=0
MOVL C01125 V=800.0 PL=0
MOVL C01126 V=800.0 PL=0
MOVL C01127 V=800.0 PL=0
MOVL C01128 V=800.0 PL=0
MOVL C01129 V=800.0 PL=0
MOVL C01130 V=800.0 PL=0
MOVL C01131 V=800.0 PL=0
MOVL C01132 V=800.0 PL=0
MOVL C01133 V=800.0 PL=0
MOVL C01134 V=800.0 PL=0
MOVL C01135 V=800.0 PL=0
MOVL C01136 V=800.0 PL=0
MOVL C01137 V=800.0 PL=0
MOVL C01138 V=800.0 PL=0
MOVL C01139 V=800.0 PL=0
MOVL C01140 V=800.0 PL=0
MOVL C01141 V=800.0 PL=0
MOVL C01142 V=800.0 PL=0
MOVL C01143 V=800.0 PL=0
MOVL C01144 V=800.0 PL=0
MOVL C01145 V=800.0 PL=0
MOVL C01146 V=800.0 PL=0
MOVL C01147 V=800.0 PL=0
MOVL C01148 V=800.0 PL=0
MOVL C01149 V=800.0 PL=0
MOVL C01150 V=800.0 PL=0
MOVL C01151 V=800.0 PL=0
MOVL C01152 V=800.0 PL=0
MOVL C01153 V=800.0 PL=0
MOVL C01154 V=800.0 PL=0
MOVL C01155 V=800.0 PL=0
MOVL C01156 V=800.0 PL=0
MOVL C01157 V=800.0 PL=0
MOVL C01158 V=800.0 PL=0
MOVL C01159 V=800.0 PL=0
MOVL C01160 V=800.0 PL=0
MOVL C01161 V=800.0 PL=0
MOVL C01162 V=800.0 PL=0
MOVL C01163 V=800.0 PL=0
MOVL C01164 V=800.0 PL=0
MOVL C01165 V=800.0 PL=0
MOVL C01166 V=800.0 PL=0
MOVL C01167 V=800.0 PL=0
MOVL C01168 V=800.0 PL=0
MOVL C01169 V=800.0 PL=0
MOVL C01170 V=800.0 PL=0
MOVL C01171 V=800.0 PL=0
MOVL C01172 V=800.0 PL=0
MOVL C01173 V=800.0 PL=0
MOVL C01174 V=800.0 PL=0
MOVL C01175 V=800.0 PL=0
MOVL C01176 V=800.0 PL=0
MOVL C01177 V=800.0 PL=0
MOVL C01178 V=800.0 PL=0
MOVL C01179 V=800.0 PL=0
MOVL C01180 V=800.0 PL=0
MOVL C01181 V=800.0 PL=0
MOVL C01182 V=800.0 PL=0
MOVL C01183 V=800.0 PL=0
MOVL C01184 V=800.0 PL=0
MOVL C01185 V=800.0 PL=0
MOVL C01186 V=800.0 PL=0
MOVL C01187 V=800.0 PL=0
MOVL C01188 V=800.0 PL=0
MOVL C01189 V=800.0 PL=0
MOVL C01190 V=800.0 PL=0
MOVL C01191 V=800.0 PL=0
MOVL C01192 V=800.0 PL=0
MOVL C01193 V=800.0 PL=0
MOVL C01194 V=800.0 PL=0
MOVL C01195 V=800.0 PL=0
MOVL C01196 V=800.0 PL=0
MOVL C01197 V=800.0 PL=0
MOVL C01198 V=800.0 PL=0
MOVL C01199 V=800.0 PL=0
MOVL C01200 V=800.0 PL=0
MOVL C01201 V=800.0 PL=0
MOVL C01202 V=800.0 PL=0
MOVL C01203 V=800.0 PL=0
MOVL C01204 V=800.0 PL=0
MOVL C01205 V=800.0 PL=0
MOVL C01206 V=800.0 PL=0
MOVL C01207 V=800.0 PL=0
MOVL C01208 V=800.0 PL=0
MOVL C01209 V=800.0 PL=0
MOVL C01210 V=800.0 PL=0
MOVL C01211 V=800.0 PL=0
MOVL C01212 V=800.0 PL=0
MOVL C01213 V=800.0 PL=0
MOVL C01214 V=800.0 PL=0
MOVL C01215 V=800.0 PL=0
MOVL C01216 V=800.0 PL=0
MOVL C01217 V=800.0 PL=0
MOVL C01218 V=800.0 PL=0
MOVL C01219 V=800.0 PL=0
MOVL C01220 V=800.0 PL=0
MOVL C01221 V=800.0 PL=0
MOVL C01222 V=800.0 PL=0
MOVL C01223 V=800.0 PL=0
MOVL C01224 V=800.0 PL=0
MOVL C01225 V=800.0 PL=0
MOVL C01226 V=800.0 PL=0
MOVL C01227 V=800.0 PL=0
MOVL C01228 V=800.0 PL=0
MOVL C01229 V=800.0 PL=0
MOVL C01230 V=800.0 PL=0
MOVL C01231 V=800.0 PL=0
MOVL C01232 V=800.0 PL=0
MOVL C01233 V=800.0 PL=0
MOVL C01234 V=800.0 PL=0
MOVL C01235 V=800.0 PL=0
MOVL C01236 V=800.0 PL=0
MOVL C01237 V=800.0 PL=0
MOVL C01238 V=800.0 PL=0
MOVL C01239 V=800.0 PL=0
MOVL C01240 V=800.0 PL=0
MOVL C01241 V=800.0 PL=0
MOVL C01242 V=800.0 PL=0
MOVL C01243 V=800.0 PL=0
MOVL C01244 V=800.0 PL=0
MOVL C01245 V=800.0 PL=0
MOVL C01246 V=800.0 PL=0
MOVL C01247 V=800.0 PL=0
MOVL C01248 V=800.0 PL=0
MOVL C01249 V=800.0 PL=0
MOVL C01250 V=800.0 PL=0
MOVL C01251 V=800.0 PL=0
MOVL C01252 V=800.0 PL=0
MOVL C01253 V=800.0 PL=0
MOVL C01254 V=800.0 PL=0
MOVL C01255 V=800.0 PL=0
MOVL C01256 V=800.0 PL=0
MOVL C01257 V=800.0 PL=0
MOVL C01258 V=800.0 PL=0
MOVL C01259 V=800.0 PL=0
MOVL C01260 V=800.0 PL=0
MOVL C01261 V=800.0 PL=0
MOVL C01262 V=800.0 PL=0
MOVL C01263 V=800.0 PL=0
MOVL C01264 V=800.0 PL=0
MOVL C01265 V=800.0 PL=0
MOVL C01266 V=800.0 PL=0
MOVL C01267 V=800.0 PL=0
MOVL C01268 V=800.0 PL=0
MOVL C01269 V=800.0 PL=0
MOVL C01270 V=800.0 PL=0
MOVL C01271 V=800.0 PL=0
MOVL C01272 V=800.0 PL=0
MOVL C01273 V=800.0 PL=0
MOVL C01274 V=800.0 PL=0
MOVL C01275 V=800.0 PL=0
MOVL C01276 V=800.0 PL=0
MOVL C01277 V=800.0 PL=0
MOVL C01278 V=800.0 PL=0
MOVL C01279 V=800.0 PL=0
MOVL C01280 V=800.0 PL=0
MOVL C01281 V=800.0 PL=0
MOVL C01282 V=800.0 PL=0
MOVL C01283 V=800.0 PL=0
MOVL C01284 V=800.0 PL=0
MOVL C01285 V=800.0 PL=0
MOVL C01286 V=800.0 PL=0
MOVL C01287 V=800.0 PL=0
MOVL C01288 V=800.0 PL=0
MOVL C01289 V=800.0 PL=0
MOVL C01290 V=800.0 PL=0
MOVL C01291 V=800.0 PL=0
MOVL C01292 V=800.0 PL=0
MOVL C01293 V=800.0 PL=0
MOVL C01294 V=800.0 PL=0
MOVL C01295 V=800.0 PL=0
MOVL C01296 V=800.0 PL=0
MOVL C01297 V=800.0 PL=0
MOVL C01298 V=800.0 PL=0
MOVL C01299 V=800.0 PL=0
MOVL C01300 V=800.0 PL=0
MOVL C01301 V=800.0 PL=0
MOVL C01302 V=800.0 PL=0
MOVL C01303 V=800.0 PL=0
MOVL C01304 V=800.0 PL=0
MOVL C01305 V=800.0 PL=0
MOVL C01306 V=800.0 PL=0
MOVL C01307 V=800.0 PL=0
MOVL C01308 V=800.0 PL=0
MOVL C01309 V=800.0 PL=0
MOVL C01310 V=800.0 PL=0
MOVL C01311 V=800.0 PL=0
MOVL C01312 V=800.0 PL=0
MOVL C01313 V=800.0 PL=0
MOVL C01314 V=800.0 PL=0
MOVL C01315 V=800.0 PL=0
MOVL C01316 V=800.0 PL=0
MOVL C01317 V=800.0 PL=0
MOVL C01318 V=800.0 PL=0
MOVL C01319 V=800.0 PL=0
MOVL C01320 V=800.0 PL=0
MOVL C01321 V=800.0 PL=0
MOVL C01322 V=800.0 PL=0
MOVL C01323 V=800.0 PL=0
MOVL C01324 V=800.0 PL=0
MOVL C01325 V=800.0 PL=0
MOVL C01326 V=800.0 PL=0
MOVL C01327 V=800.0 PL=0
MOVL C01328 V=800.0 PL=0
MOVL C01329 V=800.0 PL=0
MOVL C01330 V=800.0 PL=0
MOVL C01331 V=800.0 PL=0
MOVL C01332 V=800.0 PL=0
MOVL C01333 V=800.0 PL=0
MOVL C01334 V=800.0 PL=0
MOVL C01335 V=800.0 PL=0
MOVL C01336 V=800.0 PL=0
MOVL C01337 V=800.0 PL=0
MOVL C01338 V=800.0 PL=0
MOVL C01339 V=800.0 PL=0
MOVL C01340 V=800.0 PL=0
MOVL C01341 V=800.0 PL=0
MOVL C01342 V=800.0 PL=0
MOVL C01343 V=800.0 PL=0
MOVL C01344 V=800.0 PL=0
MOVL C01345 V=800.0 PL=0
MOVL C01346 V=800.0 PL=0
MOVL C01347 V=800.0 PL=0
MOVL C01348 V=800.0 PL=0
MOVL C01349 V=800.0 PL=0
MOVL C01350 V=800.0 PL=0
MOVL C01351 V=800.0 PL=0
MOVL C01352 V=800.0 PL=0
MOVL C01353 V=800.0 PL=0
MOVL C01354 V=800.0 PL=0
MOVL C01355 V=800.0 PL=0
MOVL C01356 V=800.0 PL=0
MOVL C01357 V=800.0 PL=0
MOVL C01358 V=800.0 PL=0
MOVL C01359 V=800.0 PL=0
MOVL C01360 V=800.0 PL=0
MOVL C01361 V=800.0 PL=0
MOVL C01362 V=800.0 PL=0
MOVL C01363 V=800.0 PL=0
MOVL C01364 V=800.0 PL=0
MOVL C01365 V=800.0 PL=0
MOVL C01366 V=800.0 PL=0
MOVL C01367 V=800.0 PL=0
MOVL C01368 V=800.0 PL=0
MOVL C01369 V=800.0 PL=0
MOVL C01370 V=800.0 PL=0
MOVL C01371 V=800.0 PL=0
MOVL C01372 V=800.0 PL=0
MOVL C01373 V=800.0 PL=0
MOVL C01374 V=800.0 PL=0
MOVL C01375 V=800.0 PL=0
MOVL C01376 V=800.0 PL=0
MOVL C01377 V=800.0 PL=0
MOVL C01378 V=800.0 PL=0
MOVL C01379 V=800.0 PL=0
MOVL C01380 V=800.0 PL=0
MOVL C01381 V=800.0 PL=0
MOVL C01382 V=800.0 PL=0
MOVL C01383 V=800.0 PL=0
MOVL C01384 V=800.0 PL=0
MOVL C01385 V=800.0 PL=0
MOVL C01386 V=800.0 PL=0
MOVL C01387 V=800.0 PL=0
MOVL C01388 V=800.0 PL=0
MOVL C01389 V=800.0 PL=0
MOVL C01390 V=800.0 PL=0
MOVL C01391 V=800.0 PL=0
MOVL C01392 V=800.0 PL=0
MOVL C01393 V=800.0 PL=0
MOVL C01394 V=800.0 PL=0
MOVL C01395 V=800.0 PL=0
MOVL C01396 V=800.0 PL=0
MOVL C01397 V=800.0 PL=0
MOVL C01398 V=800.0 PL=0
MOVL C01399 V=800.0 PL=0
MOVL C01400 V=800.0 PL=0
MOVL C01401 V=800.0 PL=0
MOVL C01402 V=800.0 PL=0
MOVL C01403 V=800.0 PL=0
MOVL C01404 V=800.0 PL=0
MOVL C01405 V=800.0 PL=0
MOVL C01406 V=800.0 PL=0
MOVL C01407 V=800.0 PL=0
MOVL C01408 V=800.0 PL=0
MOVL C01409 V=800.0 PL=0
MOVL C01410 V=800.0 PL=0
MOVL C01411 V=800.0 PL=0
MOVL C01412 V=800.0 PL=0
MOVL C01413 V=800.0 PL=0
MOVL C01414 V=800.0 PL=0
MOVL C01415 V=800.0 PL=0
MOVL C01416 V=800.0 PL=0
MOVL C01417 V=800.0 PL=0
MOVL C01418 V=800.0 PL=0
MOVL C01419 V=800.0 PL=0
MOVL C01420 V=800.0 PL=0
MOVL C01421 V=800.0 PL=0
MOVL C01422 V=800.0 PL=0
MOVL C01423 V=800.0 PL=0
MOVL C01424 V=800.0 PL=0
MOVL C01425 V=800.0 PL=0
MOVL C01426 V=800.0 PL=0
MOVL C01427 V=800.0 PL=0
MOVL C01428 V=800.0 PL=0
MOVL C01429 V=800.0 PL=0
MOVL C01430 V=800.0 PL=0
MOVL C01431 V=800.0 PL=0
MOVL C01432 V=800.0 PL=0
MOVL C01433 V=800.0 PL=0
MOVL C01434 V=800.0 PL=0
MOVL C01435 V=800.0 PL=0
MOVL C01436 V=800.0 PL=0
MOVL C01437 V=800.0 PL=0
MOVL C01438 V=800.0 PL=0
MOVL C01439 V=800.0 PL=0
MOVL C01440 V=800.0 PL=0
MOVL C01441 V=800.0 PL=0
MOVL C01442 V=800.0 PL=0
MOVL C01443 V=800.0 PL=0
MOVL C01444 V=800.0 PL=0
MOVL C01445 V=800.0 PL=0
MOVL C01446 V=800.0 PL=0
MOVL C01447 V=800.0 PL=0
MOVL C01448 V=800.0 PL=0
MOVL C01449 V=800.0 PL=0
MOVL C01450 V=800.0 PL=0
MOVL C01451 V=800.0 PL=0
MOVL C01452 V=800.0 PL=0
MOVL C01453 V=800.0 PL=0
MOVL C01454 V=800.0 PL=0
MOVL C01455 V=800.0 PL=0
MOVL C01456 V=800.0 PL=0
MOVL C01457 V=800.0 PL=0
MOVL C01458 V=800.0 PL=0
MOVL C01459 V=800.0 PL=0
MOVL C01460 V=800.0 PL=0
MOVL C01461 V=800.0 PL=0
MOVL C01462 V=800.0 PL=0
MOVL C01463 V=800.0 PL=0
MOVL C01464 V=800.0 PL=0
MOVL C01465 V=800.0 PL=0
MOVL C01466 V=800.0 PL=0
MOVL C01467 V=800.0 PL=0
MOVL C01468 V=800.0 PL=0
MOVL C01469 V=800.0 PL=0
MOVL C01470 V=800.0 PL=0
MOVL C01471 V=800.0 PL=0
MOVL C01472 V=800.0 PL=0
MOVL C01473 V=800.0 PL=0
MOVL C01474 V=800.0 PL=0
MOVL C01475 V=800.0 PL=0
MOVL C01476 V=800.0 PL=0
MOVL C01477 V=800.0 PL=0
MOVL C01478 V=800.0 PL=0
MOVL C01479 V=800.0 PL=0
MOVL C01480 V=800.0 PL=0
MOVL C01481 V=800.0 PL=0
MOVL C01482 V=800.0 PL=0
MOVL C01483 V=800.0 PL=0
MOVL C01484 V=800.0 PL=0
MOVL C01485 V=800.0 PL=0
MOVL C01486 V=800.0 PL=0
MOVL C01487 V=800.0 PL=0
MOVL C01488 V=800.0 PL=0
MOVL C01489 V=800.0 PL=0
MOVL C01490 V=800.0 PL=0
MOVL C01491 V=800.0 PL=0
MOVL C01492 V=800.0 PL=0
MOVL C01493 V=800.0 PL=0
MOVL C01494 V=800.0 PL=0
MOVL C01495 V=800.0 PL=0
MOVL C01496 V=800.0 PL=0
MOVL C01497 V=800.0 PL=0
MOVL C01498 V=800.0 PL=0
MOVL C01499 V=800.0 PL=0
MOVL C01500 V=800.0 PL=0
MOVL C01501 V=800.0 PL=0
MOVL C01502 V=800.0 PL=0
MOVL C01503 V=800.0 PL=0
MOVL C01504 V=800.0 PL=0
MOVL C01505 V=800.0 PL=0
MOVL C01506 V=800.0 PL=0
MOVL C01507 V=800.0 PL=0
MOVL C01508 V=800.0 PL=0
MOVL C01509 V=800.0 PL=0
MOVL C01510 V=800.0 PL=0
MOVL C01511 V=800.0 PL=0
MOVL C01512 V=800.0 PL=0
MOVL C01513 V=800.0 PL=0
MOVL C01514 V=800.0 PL=0
MOVL C01515 V=800.0 PL=0
MOVL C01516 V=800.0 PL=0
MOVL C01517 V=800.0 PL=0
MOVL C01518 V=800.0 PL=0
MOVL C01519 V=800.0 PL=0
MOVL C01520 V=800.0 PL=0
MOVL C01521 V=800.0 PL=0
MOVL C01522 V=800.0 PL=0
MOVL C01523 V=800.0 PL=0
MOVL C01524 V=800.0 PL=0
MOVL C01525 V=800.0 PL=0
MOVL C01526 V=800.0 PL=0
MOVL C01527 V=800.0 PL=0
MOVL C01528 V=800.0 PL=0
MOVL C01529 V=800.0 PL=0
MOVL C01530 V=800.0 PL=0
MOVL C01531 V=800.0 PL=0
MOVL C01532 V=800.0 PL=0
MOVL C01533 V=800.0 PL=0
MOVL C01534 V=800.0 PL=0
MOVL C01535 V=800.0 PL=0
MOVL C01536 V=800.0 PL=0
MOVL C01537 V=800.0 PL=0
MOVL C01538 V=800.0 PL=0
MOVL C01539 V=800.0 PL=0
MOVL C01540 V=800.0 PL=0
MOVL C01541 V=800.0 PL=0
MOVL C01542 V=800.0 PL=0
MOVL C01543 V=800.0 PL=0
MOVL C01544 V=800.0 PL=0
MOVL C01545 V=800.0 PL=0
MOVL C01546 V=800.0 PL=0
MOVL C01547 V=800.0 PL=0
MOVL C01548 V=800.0 PL=0
MOVL C01549 V=800.0 PL=0
MOVL C01550 V=800.0 PL=0
MOVL C01551 V=800.0 PL=0
MOVL C01552 V=800.0 PL=0
MOVL C01553 V=800.0 PL=0
MOVL C01554 V=800.0 PL=0
MOVL C01555 V=800.0 PL=0
MOVL C01556 V=800.0 PL=0
MOVL C01557 V=800.0 PL=0
MOVL C01558 V=800.0 PL=0
MOVL C01559 V=800.0 PL=0
MOVL C01560 V=800.0 PL=0
MOVL C01561 V=800.0 PL=0
MOVL C01562 V=800.0 PL=0
MOVL C01563 V=800.0 PL=0
MOVL C01564 V=800.0 PL=0
MOVL C01565 V=800.0 PL=0
MOVL C01566 V=800.0 PL=0
MOVL C01567 V=800.0 PL=0
MOVL C01568 V=800.0 PL=0
MOVL C01569 V=800.0 PL=0
MOVL C01570 V=800.0 PL=0
MOVL C01571 V=800.0 PL=0
MOVL C01572 V=800.0 PL=0
MOVL C01573 V=800.0 PL=0
MOVL C01574 V=800.0 PL=0
MOVL C01575 V=800.0 PL=0
MOVL C01576 V=800.0 PL=0
MOVL C01577 V=800.0 PL=0
MOVL C01578 V=800.0 PL=0
MOVL C01579 V=800.0 PL=0
MOVL C01580 V=800.0 PL=0
MOVL C01581 V=800.0 PL=0
MOVL C01582 V=800.0 PL=0
MOVL C01583 V=800.0 PL=0
MOVL C01584 V=800.0 PL=0
MOVL C01585 V=800.0 PL=0
MOVL C01586 V=800.0 PL=0
MOVL C01587 V=800.0 PL=0
MOVL C01588 V=800.0 PL=0
MOVL C01589 V=800.0 PL=0
MOVL C01590 V=800.0 PL=0
MOVL C01591 V=800.0 PL=0
MOVL C01592 V=800.0 PL=0
MOVL C01593 V=800.0 PL=0
MOVL C01594 V=800.0 PL=0
MOVL C01595 V=800.0 PL=0
MOVL C01596 V=800.0 PL=0
MOVL C01597 V=800.0 PL=0
MOVL C01598 V=800.0 PL=0
MOVL C01599 V=800.0 PL=0
MOVL C01600 V=800.0 PL=0
MOVL C01601 V=800.0 PL=0
MOVL C01602 V=800.0 PL=0
MOVL C01603 V=800.0 PL=0
MOVL C01604 V=800.0 PL=0
MOVL C01605 V=800.0 PL=0
MOVL C01606 V=800.0 PL=0
MOVL C01607 V=800.0 PL=0
MOVL C01608 V=800.0 PL=0
MOVL C01609 V=800.0 PL=0
MOVL C01610 V=800.0 PL=0
MOVL C01611 V=800.0 PL=0
MOVL C01612 V=800.0 PL=0
MOVL C01613 V=800.0 PL=0
MOVL C01614 V=800.0 PL=0
MOVL C01615 V=800.0 PL=0
MOVL C01616 V=800.0 PL=0
MOVL C01617 V=800.0 PL=0
MOVL C01618 V=800.0 PL=0
MOVL C01619 V=800.0 PL=0
MOVL C01620 V=800.0 PL=0
MOVL C01621 V=800.0 PL=0
MOVL C01622 V=800.0 PL=0
MOVL C01623 V=800.0 PL=0
MOVL C01624 V=800.0 PL=0
MOVL C01625 V=800.0 PL=0
MOVL C01626 V=800.0 PL=0
MOVL C01627 V=800.0 PL=0
MOVL C01628 V=800.0 PL=0
MOVL C01629 V=800.0 PL=0
MOVL C01630 V=800.0 PL=0
MOVL C01631 V=800.0 PL=0
MOVL C01632 V=800.0 PL=0
MOVL C01633 V=800.0 PL=0
MOVL C01634 V=800.0 PL=0
MOVL C01635 V=800.0 PL=0
MOVL C01636 V=800.0 PL=0
MOVL C01637 V=800.0 PL=0
MOVL C01638 V=800.0 PL=0
MOVL C01639 V=800.0 PL=0
MOVL C01640 V=800.0 PL=0
MOVL C01641 V=800.0 PL=0
MOVL C01642 V=800.0 PL=0
MOVL C01643 V=800.0 PL=0
MOVL C01644 V=800.0 PL=0
MOVL C01645 V=800.0 PL=0
MOVL C01646 V=800.0 PL=0
MOVL C01647 V=800.0 PL=0
MOVL C01648 V=800.0 PL=0
MOVL C01649 V=800.0 PL=0
MOVL C01650 V=800.0 PL=0
MOVL C01651 V=800.0 PL=0
MOVL C01652 V=800.0 PL=0
MOVL C01653 V=800.0 PL=0
MOVL C01654 V=800.0 PL=0
MOVL C01655 V=800.0 PL=0
MOVL C01656 V=800.0 PL=0
MOVL C01657 V=800.0 PL=0
MOVL C01658 V=800.0 PL=0
MOVL C01659 V=800.0 PL=0
MOVL C01660 V=800.0 PL=0
MOVL C01661 V=800.0 PL=0
MOVL C01662 V=800.0 PL=0
MOVL C01663 V=800.0 PL=0
MOVL C01664 V=800.0 PL=0
MOVL C01665 V=800.0 PL=0
MOVL C01666 V=800.0 PL=0
MOVL C01667 V=800.0 PL=0
MOVL C01668 V=800.0 PL=0
MOVL C01669 V=800.0 PL=0
MOVL C01670 V=800.0 PL=0
MOVL C01671 V=800.0 PL=0
MOVL C01672 V=800.0 PL=0
MOVL C01673 V=800.0 PL=0
MOVL C01674 V=800.0 PL=0
MOVL C01675 V=800.0 PL=0
MOVL C01676 V=800.0 PL=0
MOVL C01677 V=800.0 PL=0
MOVL C01678 V=800.0 PL=0
MOVL C01679 V=800.0 PL=0
MOVL C01680 V=800.0 PL=0
MOVL C01681 V=800.0 PL=0
MOVL C01682 V=800.0 PL=0
MOVL C01683 V=800.0 PL=0
MOVL C01684 V=800.0 PL=0
MOVL C01685 V=800.0 PL=0
MOVL C01686 V=800.0 PL=0
MOVL C01687 V=800.0 PL=0
MOVL C01688 V=800.0 PL=0
MOVL C01689 V=800.0 PL=0
MOVL C01690 V=800.0 PL=0
MOVL C01691 V=800.0 PL=0
MOVL C01692 V=800.0 PL=0
MOVL C01693 V=800.0 PL=0
MOVL C01694 V=800.0 PL=0
MOVL C01695 V=800.0 PL=0
MOVL C01696 V=800.0 PL=0
MOVL C01697 V=800.0 PL=0
MOVL C01698 V=800.0 PL=0
MOVL C01699 V=800.0 PL=0
MOVL C01700 V=800.0 PL=0
MOVL C01701 V=800.0 PL=0
MOVL C01702 V=800.0 PL=0
MOVL C01703 V=800.0 PL=0
MOVL C01704 V=800.0 PL=0
MOVL C01705 V=800.0 PL=0
MOVL C01706 V=800.0 PL=0
MOVL C01707 V=800.0 PL=0
MOVL C01708 V=800.0 PL=0
MOVL C01709 V=800.0 PL=0
MOVL C01710 V=800.0 PL=0
MOVL C01711 V=800.0 PL=0
MOVL C01712 V=800.0 PL=0
MOVL C01713 V=800.0 PL=0
MOVL C01714 V=800.0 PL=0
MOVL C01715 V=800.0 PL=0
MOVL C01716 V=800.0 PL=0
MOVL C01717 V=800.0 PL=0
MOVL C01718 V=800.0 PL=0
MOVL C01719 V=800.0 PL=0
MOVL C01720 V=800.0 PL=0
MOVL C01721 V=800.0 PL=0
MOVL C01722 V=800.0 PL=0
MOVL C01723 V=800.0 PL=0
MOVL C01724 V=800.0 PL=0
MOVL C01725 V=800.0 PL=0
MOVL C01726 V=800.0 PL=0
MOVL C01727 V=800.0 PL=0
MOVL C01728 V=800.0 PL=0
MOVL C01729 V=800.0 PL=0
MOVL C01730 V=800.0 PL=0
MOVL C01731 V=800.0 PL=0
MOVL C01732 V=800.0 PL=0
MOVL C01733 V=800.0 PL=0
MOVL C01734 V=800.0 PL=0
MOVL C01735 V=800.0 PL=0
MOVL C01736 V=800.0 PL=0
MOVL C01737 V=800.0 PL=0
MOVL C01738 V=800.0 PL=0
MOVL C01739 V=800.0 PL=0
MOVL C01740 V=800.0 PL=0
MOVL C01741 V=800.0 PL=0
MOVL C01742 V=800.0 PL=0
MOVL C01743 V=800.0 PL=0
MOVL C01744 V=800.0 PL=0
MOVL C01745 V=800.0 PL=0
MOVL C01746 V=800.0 PL=0
MOVL C01747 V=800.0 PL=0
MOVL C01748 V=800.0 PL=0
MOVL C01749 V=800.0 PL=0
MOVL C01750 V=800.0 PL=0
MOVL C01751 V=800.0 PL=0
MOVL C01752 V=800.0 PL=0
MOVL C01753 V=800.0 PL=0
MOVL C01754 V=800.0 PL=0
MOVL C01755 V=800.0 PL=0
MOVL C01756 V=800.0 PL=0
MOVL C01757 V=800.0 PL=0
MOVL C01758 V=800.0 PL=0
MOVL C01759 V=800.0 PL=0
MOVL C01760 V=800.0 PL=0
MOVL C01761 V=800.0 PL=0
MOVL C01762 V=800.0 PL=0
MOVL C01763 V=800.0 PL=0
MOVL C01764 V=800.0 PL=0
MOVL C01765 V=800.0 PL=0
MOVL C01766 V=800.0 PL=0
MOVL C01767 V=800.0 PL=0
MOVL C01768 V=800.0 PL=0
MOVL C01769 V=800.0 PL=0
MOVL C01770 V=800.0 PL=0
MOVL C01771 V=800.0 PL=0
MOVL C01772 V=800.0 PL=0
MOVL C01773 V=800.0 PL=0
MOVL C01774 V=800.0 PL=0
MOVL C01775 V=800.0 PL=0
MOVL C01776 V=800.0 PL=0
MOVL C01777 V=800.0 PL=0
MOVL C01778 V=800.0 PL=0
MOVL C01779 V=800.0 PL=0
MOVL C01780 V=800.0 PL=0
MOVL C01781 V=800.0 PL=0
MOVL C01782 V=800.0 PL=0
MOVL C01783 V=800.0 PL=0
MOVL C01784 V=800.0 PL=0
MOVL C01785 V=800.0 PL=0
MOVL C01786 V=800.0 PL=0
MOVL C01787 V=800.0 PL=0
MOVL C01788 V=800.0 PL=0
MOVL C01789 V=800.0 PL=0
MOVL C01790 V=800.0 PL=0
MOVL C01791 V=800.0 PL=0
MOVL C01792 V=800.0 PL=0
MOVL C01793 V=800.0 PL=0
MOVL C01794 V=800.0 PL=0
MOVL C01795 V=800.0 PL=0
MOVL C01796 V=800.0 PL=0
MOVL C01797 V=800.0 PL=0
MOVL C01798 V=800.0 PL=0
MOVL C01799 V=800.0 PL=0
MOVL C01800 V=800.0 PL=0
MOVL C01801 V=800.0 PL=0
MOVL C01802 V=800.0 PL=0
MOVL C01803 V=800.0 PL=0
MOVL C01804 V=800.0 PL=0
MOVL C01805 V=800.0 PL=0
MOVL C01806 V=800.0 PL=0
MOVL C01807 V=800.0 PL=0
MOVL C01808 V=800.0 PL=0
MOVL C01809 V=800.0 PL=0
MOVL C01810 V=800.0 PL=0
MOVL C01811 V=800.0 PL=0
MOVL C01812 V=800.0 PL=0
MOVL C01813 V=800.0 PL=0
MOVL C01814 V=800.0 PL=0
MOVL C01815 V=800.0 PL=0
MOVL C01816 V=800.0 PL=0
MOVL C01817 V=800.0 PL=0
MOVL C01818 V=800.0 PL=0
MOVL C01819 V=800.0 PL=0
MOVL C01820 V=800.0 PL=0
MOVL C01821 V=800.0 PL=0
MOVL C01822 V=800.0 PL=0
MOVL C01823 V=800.0 PL=0
MOVL C01824 V=800.0 PL=0
MOVL C01825 V=800.0 PL=0
MOVL C01826 V=800.0 PL=0
MOVL C01827 V=800.0 PL=0
MOVL C01828 V=800.0 PL=0
MOVL C01829 V=800.0 PL=0
MOVL C01830 V=800.0 PL=0
MOVL C01831 V=800.0 PL=0
MOVL C01832 V=800.0 PL=0
MOVL C01833 V=800.0 PL=0
MOVL C01834 V=800.0 PL=0
MOVL C01835 V=800.0 PL=0
MOVL C01836 V=800.0 PL=0
MOVL C01837 V=800.0 PL=0
MOVL C01838 V=800.0 PL=0
MOVL C01839 V=800.0 PL=0
MOVL C01840 V=800.0 PL=0
MOVL C01841 V=800.0 PL=0
MOVL C01842 V=800.0 PL=0
MOVL C01843 V=800.0 PL=0
MOVL C01844 V=800.0 PL=0
MOVL C01845 V=800.0 PL=0
MOVL C01846 V=800.0 PL=0
MOVL C01847 V=800.0 PL=0
MOVL C01848 V=800.0 PL=0
MOVL C01849 V=800.0 PL=0
MOVL C01850 V=800.0 PL=0
MOVL C01851 V=800.0 PL=0
MOVL C01852 V=800.0 PL=0
MOVL C01853 V=800.0 PL=0
MOVL C01854 V=800.0 PL=0
MOVL C01855 V=800.0 PL=0
MOVL C01856 V=800.0 PL=0
MOVL C01857 V=800.0 PL=0
MOVL C01858 V=800.0 PL=0
MOVL C01859 V=800.0 PL=0
MOVL C01860 V=800.0 PL=0
MOVL C01861 V=800.0 PL=0
MOVL C01862 V=800.0 PL=0
MOVL C01863 V=800.0 PL=0
MOVL C01864 V=800.0 PL=0
MOVL C01865 V=800.0 PL=0
MOVL C01866 V=800.0 PL=0
MOVL C01867 V=800.0 PL=0
MOVL C01868 V=800.0 PL=0
MOVL C01869 V=800.0 PL=0
MOVL C01870 V=800.0 PL=0
MOVL C01871 V=800.0 PL=0
MOVL C01872 V=800.0 PL=0
MOVL C01873 V=800.0 PL=0
MOVL C01874 V=800.0 PL=0
MOVL C01875 V=800.0 PL=0
MOVL C01876 V=800.0 PL=0
MOVL C01877 V=800.0 PL=0
MOVL C01878 V=800.0 PL=0
MOVL C01879 V=800.0 PL=0
MOVL C01880 V=800.0 PL=0
MOVL C01881 V=800.0 PL=0
MOVL C01882 V=800.0 PL=0
MOVL C01883 V=800.0 PL=0
MOVL C01884 V=800.0 PL=0
MOVL C01885 V=800.0 PL=0
MOVL C01886 V=800.0 PL=0
MOVL C01887 V=800.0 PL=0
MOVL C01888 V=800.0 PL=0
MOVL C01889 V=800.0 PL=0
MOVL C01890 V=800.0 PL=0
MOVL C01891 V=800.0 PL=0
MOVL C01892 V=800.0 PL=0
MOVL C01893 V=800.0 PL=0
MOVL C01894 V=800.0 PL=0
MOVL C01895 V=800.0 PL=0
MOVL C01896 V=800.0 PL=0
MOVL C01897 V=800.0 PL=0
MOVL C01898 V=800.0 PL=0
MOVL C01899 V=800.0 PL=0
MOVL C01900 V=800.0 PL=0
MOVL C01901 V=800.0 PL=0
MOVL C01902 V=800.0 PL=0
MOVL C01903 V=800.0 PL=0
MOVL C01904 V=800.0 PL=0
MOVL C01905 V=800.0 PL=0
MOVL C01906 V=800.0 PL=0
MOVL C01907 V=800.0 PL=0
MOVL C01908 V=800.0 PL=0
MOVL C01909 V=800.0 PL=0
MOVL C01910 V=800.0 PL=0
MOVL C01911 V=800.0 PL=0
MOVL C01912 V=800.0 PL=0
MOVL C01913 V=800.0 PL=0
MOVL C01914 V=800.0 PL=0
MOVL C01915 V=800.0 PL=0
MOVL C01916 V=800.0 PL=0
MOVL C01917 V=800.0 PL=0
MOVL C01918 V=800.0 PL=0
MOVL C01919 V=800.0 PL=0
MOVL C01920 V=800.0 PL=0
MOVL C01921 V=800.0 PL=0
MOVL C01922 V=800.0 PL=0
MOVL C01923 V=800.0 PL=0
MOVL C01924 V=800.0 PL=0
MOVL C01925 V=800.0 PL=0
MOVL C01926 V=800.0 PL=0
MOVL C01927 V=800.0 PL=0
MOVL C01928 V=800.0 PL=0
MOVL C01929 V=800.0 PL=0
MOVL C01930 V=800.0 PL=0
MOVL C01931 V=800.0 PL=0
MOVL C01932 V=800.0 PL=0
MOVL C01933 V=800.0 PL=0
MOVL C01934 V=800.0 PL=0
MOVL C01935 V=800.0 PL=0
MOVL C01936 V=800.0 PL=0
MOVL C01937 V=800.0 PL=0
MOVL C01938 V=800.0 PL=0
MOVL C01939 V=800.0 PL=0
MOVL C01940 V=800.0 PL=0
MOVL C01941 V=800.0 PL=0
MOVL C01942 V=800.0 PL=0
MOVL C01943 V=800.0 PL=0
MOVL C01944 V=800.0 PL=0
MOVL C01945 V=800.0 PL=0
MOVL C01946 V=800.0 PL=0
MOVL C01947 V=800.0 PL=0
MOVL C01948 V=800.0 PL=0
MOVL C01949 V=800.0 PL=0
MOVL C01950 V=800.0 PL=0
MOVL C01951 V=800.0 PL=0
MOVL C01952 V=800.0 PL=0
MOVL C01953 V=800.0 PL=0
MOVL C01954 V=800.0 PL=0
MOVL C01955 V=800.0 PL=0
MOVL C01956 V=800.0 PL=0
MOVL C01957 V=800.0 PL=0
MOVL C01958 V=800.0 PL=0
MOVL C01959 V=800.0 PL=0
MOVL C01960 V=800.0 PL=0
MOVL C01961 V=800.0 PL=0
MOVL C01962 V=800.0 PL=0
MOVL C01963 V=800.0 PL=0
MOVL C01964 V=800.0 PL=0
MOVL C01965 V=800.0 PL=0
MOVL C01966 V=800.0 PL=0
MOVL C01967 V=800.0 PL=0
MOVL C01968 V=800.0 PL=0
MOVL C01969 V=800.0 PL=0
MOVL C01970 V=800.0 PL=0
MOVL C01971 V=800.0 PL=0
MOVL C01972 V=800.0 PL=0
MOVL C01973 V=800.0 PL=0
MOVL C01974 V=800.0 PL=0
MOVL C01975 V=800.0 PL=0
MOVL C01976 V=800.0 PL=0
MOVL C01977 V=800.0 PL=0
MOVL C01978 V=800.0 PL=0
MOVL C01979 V=800.0 PL=0
MOVL C01980 V=800.0 PL=0
MOVL C01981 V=800.0 PL=0
MOVL C01982 V=800.0 PL=0
MOVL C01983 V=800.0 PL=0
MOVL C01984 V=800.0 PL=0
MOVL C01985 V=800.0 PL=0
MOVL C01986 V=800.0 PL=0
MOVL C01987 V=800.0 PL=0
MOVL C01988 V=800.0 PL=0
MOVL C01989 V=800.0 PL=0
MOVL C01990 V=800.0 PL=0
MOVL C01991 V=800.0 PL=0
MOVL C01992 V=800.0 PL=0
MOVL C01993 V=800.0 PL=0
MOVL C01994 V=800.0 PL=0
MOVL C01995 V=800.0 PL=0
MOVL C01996 V=800.0 PL=0
MOVL C01997 V=800.0 PL=0
MOVL C01998 V=800.0 PL=0
MOVL C01999 V=800.0 PL=0
MOVL C02000 V=800.0 PL=0
MOVL C02001 V=800.0 PL=0
MOVL C02002 V=800.0 PL=0
MOVL C02003 V=800.0 PL=0
MOVL C02004 V=800.0 PL=0
MOVL C02005 V=800.0 PL=0
MOVL C02006 V=800.0 PL=0
MOVL C02007 V=800.0 PL=0
MOVL C02008 V=800.0 PL=0
MOVL C02009 V=800.0 PL=0
MOVL C02010 V=800.0 PL=0
MOVL C02011 V=800.0 PL=0
MOVL C02012 V=800.0 PL=0
MOVL C02013 V=800.0 PL=0
MOVL C02014 V=800.0 PL=0
MOVL C02015 V=800.0 PL=0
MOVL C02016 V=800.0 PL=0
MOVL C02017 V=800.0 PL=0
MOVL C02018 V=800.0 PL=0
MOVL C02019 V=800.0 PL=0
MOVL C02020 V=800.0 PL=0
MOVL C02021 V=800.0 PL=0
MOVL C02022 V=800.0 PL=0
MOVL C02023 V=800.0 PL=0
MOVL C02024 V=800.0 PL=0
MOVL C02025 V=800.0 PL=0
MOVL C02026 V=800.0 PL=0
MOVL C02027 V=800.0 PL=0
MOVL C02028 V=800.0 PL=0
MOVL C02029 V=800.0 PL=0
MOVL C02030 V=800.0 PL=0
MOVL C02031 V=800.0 PL=0
MOVL C02032 V=800.0 PL=0
MOVL C02033 V=800.0 PL=0
MOVL C02034 V=800.0 PL=0
MOVL C02035 V=800.0 PL=0
MOVL C02036 V=800.0 PL=0
MOVL C02037 V=800.0 PL=0
MOVL C02038 V=800.0 PL=0
MOVL C02039 V=800.0 PL=0
MOVL C02040 V=800.0 PL=0
MOVL C02041 V=800.0 PL=0
MOVL C02042 V=800.0 PL=0
MOVL C02043 V=800.0 PL=0
MOVL C02044 V=800.0 PL=0
MOVL C02045 V=800.0 PL=0
MOVL C02046 V=800.0 PL=0
MOVL C02047 V=800.0 PL=0
MOVL C02048 V=800.0 PL=0
MOVL C02049 V=800.0 PL=0
MOVL C02050 V=800.0 PL=0
MOVL C02051 V=800.0 PL=0
MOVL C02052 V=800.0 PL=0
MOVL C02053 V=800.0 PL=0
MOVL C02054 V=800.0 PL=0
MOVL C02055 V=800.0 PL=0
MOVL C02056 V=800.0 PL=0
MOVL C02057 V=800.0 PL=0
MOVL C02058 V=800.0 PL=0
MOVL C02059 V=800.0 PL=0
MOVL C02060 V=800.0 PL=0
MOVL C02061 V=800.0 PL=0
MOVL C02062 V=800.0 PL=0
MOVL C02063 V=800.0 PL=0
MOVL C02064 V=800.0 PL=0
MOVL C02065 V=800.0 PL=0
MOVL C02066 V=800.0 PL=0
MOVL C02067 V=800.0 PL=0
MOVL C02068 V=800.0 PL=0
MOVL C02069 V=800.0 PL=0
MOVL C02070 V=800.0 PL=0
MOVL C02071 V=800.0 PL=0
MOVL C02072 V=800.0 PL=0
MOVL C02073 V=800.0 PL=0
MOVL C02074 V=800.0 PL=0
MOVL C02075 V=800.0 PL=0
MOVL C02076 V=800.0 PL=0
MOVL C02077 V=800.0 PL=0
MOVL C02078 V=800.0 PL=0
MOVL C02079 V=800.0 PL=0
MOVL C02080 V=800.0 PL=0
MOVL C02081 V=800.0 PL=0
MOVL C02082 V=800.0 PL=0
MOVL C02083 V=800.0 PL=0
MOVL C02084 V=800.0 PL=0
MOVL C02085 V=800.0 PL=0
MOVL C02086 V=800.0 PL=0
MOVL C02087 V=800.0 PL=0
MOVL C02088 V=800.0 PL=0
MOVL C02089 V=800.0 PL=0
MOVL C02090 V=800.0 PL=0
MOVL C02091 V=800.0 PL=0
MOVL C02092 V=800.0 PL=0
MOVL C02093 V=800.0 PL=0
MOVL C02094 V=800.0 PL=0
MOVL C02095 V=800.0 PL=0
MOVL C02096 V=800.0 PL=0
MOVL C02097 V=800.0 PL=0
MOVL C02098 V=800.0 PL=0
MOVL C02099 V=800.0 PL=0
MOVL C02100 V=800.0 PL=0
MOVL C02101 V=800.0 PL=0
MOVL C02102 V=800.0 PL=0
MOVL C02103 V=800.0 PL=0
MOVL C02104 V=800.0 PL=0
MOVL C02105 V=800.0 PL=0
MOVL C02106 V=800.0 PL=0
MOVL C02107 V=800.0 PL=0
MOVL C02108 V=800.0 PL=0
